(* CODESYS project sensata_utilities.library
   Company: Sensata Technologies
   Version: 1.0.2
   DocFormat: reStructuredText
   Placeholder: Sensata_Utilities
   Title: Sensata_Utilities

Project tree, tasks and I/O mapping:
  libraries: Sensata_Common, * (Sensata Technologies); Tc2_ModbusRTU, * (Beckhoff Automation GmbH); Tc2_ModbusSrv, * (Beckhoff Automation GmbH); Tc2_SerialCom, * (Beckhoff Automation GmbH); Tc2_Standard, * (Beckhoff Automation GmbH); Tc2_System, * (Beckhoff Automation GmbH); Tc2_Utilities, * (Beckhoff Automation GmbH); Tc3_JsonXml, * (Beckhoff Automation GmbH); Tc3_Module, * (Beckhoff Automation GmbH)
  Abstract/
    Obsolete/
      function block FB_DeviceAPI [ST]: M_Connect, M_Disconnect, M_GetConnectStatus, P_bConnectBusy, P_bConnected, M_CallMethod, M_GetProperty, P_bDeviceInterfaceBusy
    function block FB_CommandRouter [ST]: M_Connect, M_Disconnect, M_GetConnectStatus, P_bConnectBusy, P_bConnected, M_AwaitCommand, M_RequestRoute, M_RouteCommand, P_bCommandRoutingBusy
    function block FB_Modbus [ST]: M_Diagnostics, M_ReadCoils, M_ReadInputRegs, M_ReadInputStatus, M_ReadRegs, M_WriteMultipleCoils, M_WriteRegs, M_WriteSingleCoil, M_WriteSingleRegister, P_bModbusBusy
    function block FB_ResourceManager [ST]: M_Reset, P_bResetBusy, M_CheckIn, M_CheckOut, P_bCheckedOut, P_strCheckedOutBy
  Concrete/
    API/
      Obsolete/
        function block FB_AdsDeviceAPI [ST]: M_CallMethod, M_GetProperty, P_bDeviceInterfaceBusy
      data type E_ApiDeviceError
      function block FB_AdsCommandRouter [ST]: M_BuildMessage, M_ParseResult, M_RouteCommand, P_bCommandRoutingBusy
      function block FB_ApiDeviceTemplate [ST]: M_Abort, P_bAbortBusy, M_Connect, M_Disconnect, M_GetConnectStatus, P_bConnectBusy, P_bConnected, M_Disable, M_Enable, M_GetEnableStatus, P_bEnableBusy, P_bEnabled, M_GetPowerStatus, M_PowerOff, M_PowerOn, P_bPowerBusy, P_bPoweredOn, M_GetCurrentProgram, M_GetProgramState, M_LoadProgram, M_PauseProgram, M_StartProgram, M_StopProgram, P_bProgramControlBusy, P_enumProgramState, P_strCurrentProgram, M_Reset, P_bResetBusy, A_CommandRecovery, M_CommandTemplate, M_RouterHelper
      function block FB_ApiParamBuilder [ST]: M_AddArrayElement, M_AddEmptyArray, M_AddEmptyArrayToArray, M_AddEmptyArrayToStruct, M_AddEmptyStruct, M_AddEmptyStructToArray, M_AddEmptyStructToStruct, M_AddParameter, M_AddStructMember, M_ClearParameters, M_OutputToParameterList, M_Add, M_Pushback, M_ParseBool, M_ParseDateTime, M_ParseDouble, M_ParseInt, M_ParseInt64, M_ParseString, M_ParseUint, M_ParseUint64, M_GetArrayElement, M_GetParameter, M_GetStructMember, M_LoadFromParameterList
    IO Mapping/
      Obsolete/
        function F_LinkDigitalIOStructs [ST]
        function F_SetDigitalInput [ST]
        function F_SetDigitalOutput [ST]
        data type ST_DebugDigitalIO
      function F_LinkDigitalIO [ST]
      function F_SetDigitalIO [ST]
      data type ST_DigitalIO
    Light Control/
      function block FB_PackMLIndicators [ST]
    Modbus/
      function block FB_ModbusMasterRTU [ST]: M_Diagnostics, M_ReadCoils, M_ReadInputRegs, M_ReadInputStatus, M_ReadRegs, M_WriteMultipleCoils, M_WriteRegs, M_WriteSingleCoil, M_WriteSingleRegister, P_bModbusBusy, A_CommandRecovery
      function block FB_ModbusTCPClient [ST]: M_Diagnostics, M_ReadCoils, M_ReadInputRegs, M_ReadInputStatus, M_ReadRegs, M_WriteMultipleCoils, M_WriteRegs, M_WriteSingleCoil, M_WriteSingleRegister, P_bModbusBusy, A_CommandRecovery
    Resource Manager/
      function block FB_FifoBufferResMgr [ST]: M_Reset, P_bResetBusy, M_CheckIn, M_CheckOut, P_bCheckedOut, P_strCheckedOutBy
  DUTs/
    Obsolete/
      data type T_ApiMethodParameters
    data type E_AdsCommandRouterError
    data type ST_ApiParameter
    data type T_ApiMessage
    data type T_ApiParameterList
    data type T_ApiParamValue
  Functions/
    function F_ButtonToggle [ST]
    function F_CalcCycleTime [ST]
  Globals/
    Obsolete/
      global variables GVL_DeviceAPI
    global variables GVL_Api
  Interfaces/
    Obsolete/
      interface I_DeviceInterface: M_CallMethod, M_GetProperty, P_bDeviceInterfaceBusy
      interface I_ModularAPI: M_CallMethod, P_bApiBusy
    interface I_CommandRouting: M_AwaitCommand, M_RequestRoute, M_RouteCommand, P_bCommandRoutingBusy
    interface I_Modbus: M_ReadCoils, M_ReadInputRegs, M_ReadInputStatus, M_ReadRegs, M_WriteMultipleCoils, M_WriteRegs, M_WriteSingleCoil, M_WriteSingleRegister, P_bModbusBusy
    interface I_ResourceManagement: M_CheckIn, M_CheckOut, P_bCheckedOut, P_strCheckedOutBy
  Project Information/
    function F_GetCompany [ST]
    function F_GetTitle [ST]
    function F_GetVersion [ST]
  Version/
    global variables Global_Version
*)

// Concrete/API/E_ApiDeviceError
{attribute 'qualified_only'}
{attribute 'strict'}
TYPE E_ApiDeviceError :
(
	None := 0,
	
	CommandRouterError			:= 0100, // Error on the command router FB
	CommandFault 				:= 0101, // Command failed to execute
	
	FailedToConnect 			:= 0200, // Connect command failed
	FailedToDisconnect 			:= 0201, // Disonnect command failed
	FailedToGetConnectStatus 	:= 0202, // GetConnectStatus command failed
	
	FailedToLoadProgram			:= 0300, // LoadProgram command failed
	FailedToGetCurrentProgram	:= 0301, // GetCurrentProgram command failed
	FailedToStartProgram		:= 0302, // StartProgram command failed
	FailedToStopProgram			:= 0303, // StopProgram command failed
	FailedToPauseProgram		:= 0304, // PauseProgram command failed
	FailedToGetProgramState		:= 0305, // GetProgramState command failed
	
	FailedToEnable				:= 0400, // Enable command failed
	FailedToDisable				:= 0401, // Disable command failed
	FailedToGetEnableStatus		:= 0402, // GetEnableStatus command failed
	
	FailedToPowerOn				:= 0500, // PowerOn command failed
	FailedToPowerOff			:= 0501, // PowerOff command failed
	FailedToGetPowerStatus		:= 0502, // GetPowerStatus command failed
	
	FailedToReset				:= 0600, // Reset command failed

	FailedToAbort				:= 0700  // Abort command failed
) UDINT;
END_TYPE

// Concrete/IO Mapping/Obsolete/ST_DebugDigitalIO
{attribute 'obsolete' := 'Use ST_DigitalIO instead.'} 
TYPE ST_DebugDigitalIO :
STRUCT
	(* Label for this IO. *)
	strLabel: T_MaxString;
	(* Current value. *)
	bCurrentValue: BOOL;
	(* Set to TRUE if IO is an output. *)
	bOutput: BOOL;
	(* Set TRUE to force output to a value. *)
	bForce: BOOL;
	(* Value to force output to. *)
	bForceValue: BOOL;
END_STRUCT
END_TYPE

// Concrete/IO Mapping/ST_DigitalIO
TYPE ST_DigitalIO :
STRUCT
	(* Device this digital IO is physically connected to e.g. 'BR-100'*)
	strDevice: T_MaxString;
	(* Address of this digital IO e.g. 'Y1224' for output 1224. *)
	strAddress: T_MaxString;
	(* Label for this digital IO in English e.g. 'Tooling Down Cylinder' *)
	strLabel: T_MaxString;
	(* ID for the label for use with language switching. *)
	udintLabelId: UDINT;
	(* Current value of the digital IO. *)
	bValue: BOOL;
	(* Value to force the value to. *)
	bForceValue: BOOL;
	(* TRUE if the value is being forced. *)
	bForced: BOOL;
END_STRUCT
END_TYPE

// DUTs/Obsolete/T_ApiMethodParameters
{attribute 'obsolete' := 'Only used on obsolete FB_DeviceAPI'} 
TYPE T_ApiMethodParameters : 
	ARRAY [1..GVL_DeviceAPI.uintMAX_CALL_METHOD_PARAMETERS]
		OF ARRAY [1..2] OF Tc2_System.T_MaxString;
END_TYPE

// DUTs/E_AdsCommandRouterError
{attribute 'qualified_only'}
{attribute 'strict'}
TYPE E_AdsCommandRouterError :
(
	None := 0,
	IncorrectResponseFormat := 100,
	NoResponseReceived := 101,
	AdsError := 200,
	PointerError := 300
) UDINT;
END_TYPE

// DUTs/ST_ApiParameter
TYPE ST_ApiParameter :
STRUCT
	strKey : T_MaxString;
	strValue : T_ApiParamValue;
END_STRUCT
END_TYPE

// DUTs/T_ApiMessage
TYPE T_ApiMessage : STRING(GVL_Api.dintMSG_STRING_SIZE); END_TYPE

// DUTs/T_ApiParameterList
TYPE T_ApiParameterList : ARRAY[GVL_Api.dintPARAM_LOWER_BOUND..GVL_Api.dintPARAM_UPPER_BOUND] OF ST_ApiParameter; END_TYPE

// DUTs/T_ApiParamValue
TYPE T_ApiParamValue : STRING(GVL_Api.dintPARAM_STRING_SIZE); END_TYPE

// Globals/Obsolete/GVL_DeviceAPI
{attribute 'qualified_only'}
VAR_GLOBAL CONSTANT
	uintMAX_CALL_METHOD_PARAMETERS : UINT := 16;
END_VAR

// Globals/GVL_Api
{attribute 'qualified_only'}
VAR_GLOBAL CONSTANT
	dintPARAM_LOWER_BOUND : DINT := 0;
	dintPARAM_UPPER_BOUND : DINT := 31;
	dintPARAM_STRING_SIZE : DINT := 1023;
	dintMSG_STRING_SIZE : DINT := 4095;
END_VAR

// Version/Global_Version
{attribute 'TcGenerated'}
{attribute 'no-analysis'}
{attribute 'linkalways'}
// This function has been automatically generated from the project information.
VAR_GLOBAL CONSTANT
	{attribute 'const_non_replaced'}
	stLibVersion_Sensata_Utilities : ST_LibVersion := (iMajor := 1, iMinor := 0, iBuild := 2, iRevision := 0, nFlags := 0, sVersion := '1.0.2');
END_VAR

// Abstract/Obsolete/FB_DeviceAPI
(*
===============================================================================
Abstract Device API
===============================================================================
:Contact: Kevin Sanita <ksanita@sensata.com>
:Last Edited: March 2022

:Description: Represents a device API that allows for methods and
	properties to be called and accessed

:Notes:
* ``M_CallMethod`` to send a call method command to a device API
* ``M_GetProperty`` to send a get property command to a device API

:Change Log:
- **March 25, 2022** Initial version
*)
{attribute 'obsolete' := 'Use FB_CommandRouter instead!'} 
FUNCTION_BLOCK ABSTRACT FB_DeviceAPI EXTENDS FB_Module IMPLEMENTS I_DeviceInterface, I_Connectable
VAR_INPUT
END_VAR
VAR_OUTPUT
END_VAR
VAR
	bConnected: BOOL;
END_VAR

(* Connect to the device. *)
METHOD M_Connect : BOOL
bConnected := TRUE;
M_Connect := TRUE;
THIS^.M_LogWarning('M_Connect not implemented!');
END_METHOD

(* Disconnect from the camera. *)
METHOD M_Disconnect : BOOL
bConnected := FALSE;
M_Disconnect := TRUE;
THIS^.M_LogWarning('M_Disconnect not implemented!');
END_METHOD

(* Get the device connection status. *)
METHOD M_GetConnectStatus : BOOL
VAR_OUTPUT
	(* TRUE if the device is connected, FALSE otherwise. *)
	bConnected	: BOOL;
END_VAR
bConnected := THIS^.bConnected;
M_GetConnectStatus := TRUE;
END_METHOD

(* TRUE while the device is connecting or disconnecting. *)
PROPERTY P_bConnectBusy : BOOL
GET
P_bConnectBusy := FALSE;
END_GET
END_PROPERTY

(* TRUE if the camera is connected. *)
PROPERTY P_bConnected : BOOL
GET
P_bConnected := bConnected;
END_GET
END_PROPERTY

(* Calls a device method from a device API. *)
METHOD M_CallMethod : BOOL
VAR_INPUT
	(* UniqueID of the target module. *)
	strTargetId		: Tc2_System.T_MaxString;
	(* Name of the method to call. *)
	strMethodName	: Tc2_System.T_MaxString;
	(* 2D array of parameter name and parameter value. *)
	arrParameters	: T_ApiMethodParameters;
END_VAR
VAR_OUTPUT
	(* Return data of the method. *)
	strReturn	: Tc2_System.T_MaxString;
END_VAR
M_CallMethod := FALSE;
END_METHOD

(* Gets the value of a device property through an API. *)
METHOD M_GetProperty : BOOL
VAR_INPUT
	(* Name of the property to get. *)
	strPropertyName	: Tc2_System.T_MaxString;
END_VAR
VAR_OUTPUT
	(* Value of the property. *)
	strReturn	: Tc2_System.T_MaxString;
END_VAR
M_GetProperty := FALSE;
END_METHOD

(* True while a device interface command is running. *)
PROPERTY P_bDeviceInterfaceBusy : BOOL
GET
P_bDeviceInterfaceBusy := FALSE;
END_GET
END_PROPERTY

END_FUNCTION_BLOCK

// Abstract/FB_CommandRouter
FUNCTION_BLOCK FB_CommandRouter EXTENDS FB_Module
	IMPLEMENTS I_CommandRouting, I_Connectable
VAR_INPUT
END_VAR
VAR_OUTPUT
END_VAR
VAR
	cr_bConnected: BOOL;
END_VAR

(* This method should establish any external connections required to use the
	functions of the device, and return TRUE and set P_bConnected to TRUE once
	connected. *)
METHOD M_Connect : BOOL
THIS^.M_LogWarning('M_Connect not implemented!');
cr_bConnected := TRUE;
M_Connect := TRUE;
END_METHOD

(* This method should break any connections established by M_Connect. It should
	immediately set P_bConnected to false unless all connections are known to
	be still active, and return TRUE once those connections are all fully
	disconnected. *)
METHOD M_Disconnect : BOOL
THIS^.M_LogWarning('M_Disconnect not implemented!');
cr_bConnected := FALSE;
M_Disconnect := TRUE;
END_METHOD

(* This method should explicitly check the connection status of the device.
	Once the connection status is known, this method should return TRUE.
	If this method fails, P_bConnected should be set to FALSE since the device
	is not absolutely known to still be connected. *)
METHOD M_GetConnectStatus : BOOL
VAR_OUTPUT
	(* This should return TRUE if all connections required to make the device
		function properly are known to be connected, and FALSE otherwise. *)
	bConnected	: BOOL;
END_VAR
THIS^.M_LogWarning('M_GetConnectStatus not implemented!');
M_GetConnectStatus := TRUE;
bConnected := cr_bConnected;
END_METHOD

(* This property should be TRUE while any method in this interface is actively
	executing, or FALSE otherwise. *)
PROPERTY P_bConnectBusy : BOOL
GET
P_bConnectBusy := FALSE;
END_GET
END_PROPERTY

(* This should be set to TRUE if M_Connect is successful or M_GetConnectStatus
	determines the device to be connected, and set to FALSE if M_Disconnect is
	called at all, M_GetConnectStatus fails, or M_GetConnectStatus determines
	the device to be not connected. *)
PROPERTY P_bConnected : BOOL
GET
P_bConnected := cr_bConnected;
END_GET
END_PROPERTY

(* Waits for the command with the given route ID to complete. *)
METHOD M_AwaitCommand : BOOL
VAR_INPUT
	(* ID assigned to the route. *)
	_in_udintRouteId	: UDINT;
	(* Timeout time for the command. *)
	_in_timeTimeout	: TIME;
END_VAR
VAR_IN_OUT
	(* Array of data key:value pairs. This will be filled with output
		data on command success. This is required due to memory limitations
		within Beckhoff. *)
	_inout_arrOutputs	: T_ApiParameterList;
END_VAR
VAR_OUTPUT
	(* True if the command executed without error. Does not necessarily
	mean the command performed the task it was expected to perform, just
	means that the method returned a value. *)
	_out_bCommandExecuted	: BOOL;
	(* The return value of the method. *)
	_out_strReturnValue	: T_ApiParamValue;
END_VAR
THIS^.M_LogWarning('M_AwaitCommand not implemented!');
M_AwaitCommand := TRUE;
END_METHOD

(* Sends a route request and returns a route ID if successfully routed. 
Use M_AwaitCommand with the route ID as input in order to wait for and get
the results of the routed command. *)
METHOD M_RequestRoute : BOOL
VAR_INPUT
	(* Unique ID of the module to call the command on. *)
	_in_strModuleId	: Tc2_System.T_MaxString;
	(* Name of the method to call. *)
	_in_strMethodName	: Tc2_System.T_MaxString;
	(* Timeout time for the route. *)
	_in_timeTimeout	: TIME;
END_VAR
VAR_IN_OUT
	(* Array of data key:value pairs. This should be set to the parameters
		of the command. *)
	_inout_arrParameters	: T_ApiParameterList;
END_VAR
VAR_OUTPUT
	(* ID assigned to the route. *)
	_out_udintRouteId	: UDINT;
END_VAR
THIS^.M_LogWarning('M_RequestRoute not implemented!');
M_RequestRoute := TRUE;
END_METHOD

(* Routes the given command and waits for the command to finish before
returning the output data of the command. *)
METHOD M_RouteCommand : BOOL
VAR_INPUT
	(* Unique ID of the module to call the command on. *)
	_in_strModuleId	: Tc2_System.T_MaxString;
	(* Name of the method to call. *)
	_in_strMethodName	: Tc2_System.T_MaxString;
	(* Timeout time for the command. *)
	_in_timeTimeout	: TIME;
END_VAR
VAR_IN_OUT
	(* Array of input parameter key:value pairs. *)
	_inout_arrParameters	: T_ApiParameterList;
	(* Array of output key:value pairs. Will be cleared and then populated with output data. *)
	_inout_arrOutputs	: T_ApiParameterList;
END_VAR
VAR_OUTPUT
	(* True if the command executed without error. Does not necessarily
	mean the command performed the task it was expected to perform, just
	means that the method returned a value. *)
	_out_bCommandExecuted	: BOOL;
	(* The return value of the method as a string. *)
	_out_strReturnValue	: T_ApiParamValue;
END_VAR
THIS^.M_LogWarning('M_RouteCommand not implemented!');
M_RouteCommand := TRUE;
END_METHOD

(* TRUE while any method in this interface is running. *)
PROPERTY P_bCommandRoutingBusy : BOOL
GET
P_bCommandRoutingBusy := TRUE;
END_GET
END_PROPERTY

END_FUNCTION_BLOCK

// Interfaces/I_CommandRouting
INTERFACE I_CommandRouting

(* Waits for the command with the given route ID to complete. *)
METHOD M_AwaitCommand : BOOL
VAR_INPUT
	(* ID assigned to the route. *)
	_in_udintRouteId : UDINT;
	
	(* Timeout time for the command. *)
	_in_timeTimeout : TIME;
END_VAR
VAR_IN_OUT
	(* Array of data key:value pairs. This will be filled with output
		data on command success. This is required due to memory limitations
		within Beckhoff. *)
	_inout_arrOutputs : T_ApiParameterList;
END_VAR
VAR_OUTPUT
	(* True if the command executed without error. Does not necessarily
	mean the command performed the task it was expected to perform, just
	means that the method returned a value. *)
	_out_bCommandExecuted : BOOL;
	
	(* The return value of the method. *)
	_out_strReturnValue : T_ApiParamValue;
END_VAR
END_METHOD

(* Sends a route request and returns a route ID if successfully routed. 
Use M_AwaitCommand with the route ID as input in order to wait for and get
the results of the routed command. *)
METHOD M_RequestRoute : BOOL
VAR_INPUT
	(* Unique ID of the module to call the command on. *)
	_in_strModuleId : T_MaxString;
	
	(* Name of the method to call. *)
	_in_strMethodName : T_MaxString;
	
	(* Timeout time for the route. *)
	_in_timeTimeout : TIME;
END_VAR
VAR_IN_OUT
	(* Array of data key:value pairs. This should be set to the parameters
		of the command. *)
	_inout_arrParameters : T_ApiParameterList;
END_VAR
VAR_OUTPUT
	(* ID assigned to the route. *)
	_out_udintRouteId : UDINT;
END_VAR
END_METHOD

(* Routes the given command and waits for the command to finish before
returning the output data of the command. *)
METHOD M_RouteCommand : BOOL
VAR_INPUT
	(* Unique ID of the module to call the command on. *)
	_in_strModuleId	: Tc2_System.T_MaxString;
	
	(* Name of the method to call. *)
	_in_strMethodName	: Tc2_System.T_MaxString;
	
	(* Timeout time for the command. *)
	_in_timeTimeout	: TIME;
END_VAR
VAR_IN_OUT
	(* Array of input parameter key:value pairs. *)
	_inout_arrParameters	: T_ApiParameterList;
	
	(* Array of output key:value pairs. Will be cleared and then populated with output data. *)
	_inout_arrOutputs	: T_ApiParameterList;
END_VAR
VAR_OUTPUT
	(* True if the command executed without error. Does not necessarily
	mean the command performed the task it was expected to perform, just
	means that the method returned a value. *)
	_out_bCommandExecuted	: BOOL;
	
	(* The return value of the method as a string. *)
	_out_strReturnValue	: T_ApiParamValue;
END_VAR
END_METHOD

(* TRUE while any method in this interface is running. *)
PROPERTY P_bCommandRoutingBusy : BOOL
GET
END_GET
END_PROPERTY

END_INTERFACE

// Interfaces/Obsolete/I_DeviceInterface
INTERFACE I_DeviceInterface

(* Calls a device method from a device API. *)
METHOD M_CallMethod : BOOL
VAR_INPUT
	(* UniqueID of the target module. *)
	strTargetId		: Tc2_System.T_MaxString;
		
	(* Name of the method to call. *)
	strMethodName : T_MaxString;
	
	(* 2D array of parameter name and parameter value. *)
	arrParameters : T_ApiMethodParameters;
END_VAR
VAR_OUTPUT
	(* Return data of the method. *)
	strReturn : T_MaxString;
END_VAR
END_METHOD

(* Gets the value of a device property through an API. *)
METHOD M_GetProperty : BOOL
VAR_INPUT
	(* Name of the property to get. *)
	strPropertyName : T_MaxString;
END_VAR
VAR_OUTPUT
	(* Value of the property. *)
	strReturn : T_MaxString;
END_VAR
END_METHOD

(* True while a device interface command is running. *)
PROPERTY P_bDeviceInterfaceBusy : BOOL
GET
END_GET
END_PROPERTY

END_INTERFACE

// Abstract/FB_Modbus
FUNCTION_BLOCK ABSTRACT FB_Modbus EXTENDS FB_Module
	IMPLEMENTS I_Modbus
VAR_INPUT
END_VAR
VAR_OUTPUT
END_VAR
VAR
END_VAR

(* Modbus Function Code 8 = Diagnostic *)
(* The diagnosis function provides a series of tests for checking the communication 
system between the master and the slave and for examining a variety of internal 
error states within the slave *)
METHOD M_Diagnostics : BOOL
VAR_INPUT
	(* Timeout value for waiting for a response from the addressed slave *)
	_in_timeTimeout : TIME;	
END_VAR
VAR_OUTPUT
	(* Contains the number of bytes currently read *)
	_out_udintcbRead : UDINT;
END_VAR
M_Diagnostics := TRUE;
THIS^.M_LogWarning('M_Diagnostics not implemented!');
END_METHOD

(* Modbus Function Code 1 = Read Coils *)
(* This function is used for reading 1 to 2048 digital outputs (coils.
One digital output corresponds to one bit of the read data bytes. *)
METHOD M_ReadCoils : BOOL
VAR_INPUT
	(* Number of data words to be read or written for word-oriented Modbus functions. For bit-oriented Modbus functions, Quantity specifies the number of bits (inputs or coils) *)
	_in_wordQuantity : WORD;
	(* Modbus Data Address from which the data are read from the end device(slave) *)
	_in_wordMBAddr : WORD;
	(* Size of the data variable used for send or read actions in bytes *)
	_in_udintcbLength : UDINT;
	(* pDestAddr for Modbus TCP FB_MBReadCoils*)
	_in_bytepMemoryAddr	: POINTER TO BYTE;
	(* Timeout value for waiting for a response from the addressed slave *)
	_in_timeTimeout	: TIME;
END_VAR
VAR_OUTPUT
	(* Contains the number of bytes currently read *)
	_out_udintcbRead : UDINT;
END_VAR
M_ReadCoils := TRUE;
THIS^.M_LogWarning('M_ReadCoils not implemented!');
END_METHOD

(* Modbus Function Code 4 = Read Input Registers *)
(* This function is used for reading 1 to 128 output registers (16 bit.
The first byte contains the lower eight bits and the second byte the upper eight bits. *)
METHOD M_ReadInputRegs : BOOL
VAR_INPUT
	(* Number of data words to be read or written for word-oriented Modbus functions. For bit-oriented Modbus functions, Quantity specifies the number of bits (inputs or coils) *)
	_in_wordQuantity : WORD;
	(* Modbus Data Address from which the data are read from the end device(slave) *)
	_in_wordMBAddr : WORD;
	(* Size of the data variable used for send or read actions in bytes *)
	_in_udintcbLength : UDINT;
	(* pDestAddr for Modbus TCP FB_MBReadInputRegs*)
	_in_bytepMemoryAddr : POINTER TO BYTE;
	(* Timeout value for waiting for a response from the addressed slave *)
	_in_timeTimeout : TIME;
END_VAR
VAR_OUTPUT
	(* Contains the number of bytes currently read *)
	_out_udintcbRead : UDINT;
END_VAR
M_ReadInputRegs := TRUE;
THIS^.M_LogWarning('M_ReadInputRegs not implemented!');
END_METHOD

(* Modbus Function Code 2 = Read Discrete Inputs *)
(* This function is used for reading 1 to 2048 digital inputs. One digital input 
corresponds to one bit of the read data bytes *)
METHOD M_ReadInputStatus : BOOL (* FB_MBReadInputs for Modbus TCP*)
VAR_INPUT
	(* Number of data words to be read or written for word-oriented Modbus functions. For bit-oriented Modbus functions, Quantity specifies the number of bits (inputs or coils) *)
	_in_wordQuantity : WORD;
	(* Modbus Data Address from which the data are read from the end device(slave) *)
	_in_wordMBAddr	: WORD;
	(* Size of the data variable used for send or read actions in bytes *)
	_in_udintcbLength : UDINT;
	(* pDestAddr for Modbus TCP FB_MBReadInputs*)
	_in_bytepMemoryAddr	: POINTER TO BYTE;
	(* Timeout value for waiting for a response from the addressed slave *)
	_in_timeTimeout	: TIME;
END_VAR
VAR_OUTPUT
	(* Contains the number of bytes currently read *)
	_out_udintcbRead : UDINT;
END_VAR
M_ReadInputStatus := TRUE;
THIS^.M_LogWarning('M_ReadInputStatus not implemented!');
END_METHOD

(* Modbus Function Code 3 = Read Registers *)
(* This function is used for reading 1 to 128 output registers (16 bit). 
The first byte contains the lower eight bits and the second byte the upper eight bits. *)
METHOD M_ReadRegs : BOOL
VAR_INPUT
	(* Number of data words to be read or written for word-oriented Modbus functions. For bit-oriented Modbus functions, Quantity specifies the number of bits (inputs or coils) *)
	_in_wordQuantity : WORD;
	(* Modbus Data Address from which the data are read from the end device(slave) *)
	_in_wordMBAddr : WORD;
	(* Size of the data variable used for send or read actions in bytes *)
	_in_udintcbLength : UDINT;
	(* pDestAddr for Modbus TCP FB_MBReadRegs*)
	_in_bytepMemoryAddr	: POINTER TO BYTE;
	(* Timeout value for waiting for a response from the addressed slave *)
	_in_timeTimeout	: TIME;
END_VAR
VAR_OUTPUT
	(* Contains the number of bytes currently read *)
	_out_udintcbRead : UDINT;
END_VAR
M_ReadRegs := TRUE;
THIS^.M_LogWarning('M_ReadRegs not implemented!');
END_METHOD

(* Modbus Function Code 15 = Write Multiple Coils *)
(* This function is used for writing 1 to 2048 digital outputs (coils). 
One digital output corresponds to one bit of the write data bytes *)
METHOD M_WriteMultipleCoils : BOOL (* FB_MBWriteCoils for Modbus TCP*)
VAR_INPUT
	(* Number of data words to be read or written for word-oriented Modbus functions. For bit-oriented Modbus functions, Quantity specifies the number of bits (inputs or coils) *)
	_in_wordQuantity : WORD;
	(* Modbus Data Address from which the data are read from the end device(slave) *)
	_in_wordMBAddr : WORD;
	(* Size of the data variable used for send or read actions in bytes *)
	_in_udintcbLength : UDINT;
	(* pDestAddr for Modbus TCP FB_MBReadCoils*)
	_in_bytepMemoryAddr	: POINTER TO BYTE;
	(* Timeout value for waiting for a response from the addressed slave *)
	_in_timeTimeout	: TIME;
END_VAR
M_WriteMultipleCoils := TRUE;
THIS^.M_LogWarning('M_WriteMultipleCoils not implemented!');
END_METHOD

(* Modbus Function Code 16 = Write Registers *)
(* This function is used for writing 1 to 128 output registers (16 bit). *)
METHOD M_WriteRegs : BOOL
VAR_INPUT
	(* Number of data words to be read or written for word-oriented Modbus functions. For bit-oriented Modbus functions, Quantity specifies the number of bits (inputs or coils) *)
	_in_wordQuantity : WORD;
	(* Modbus Data Address from which the data are read from the end device(slave) *)
	_in_wordMBAddr	: WORD;
	(* Size of the data variable used for send or read actions in bytes *)
	_in_udintcbLength : UDINT;
	(* pDestAddr for Modbus TCP FB_MBWriteRegs*)
	_in_bytepMemoryAddr	: POINTER TO BYTE;
	(* Timeout value for waiting for a response from the addressed slave *)
	_in_timeTimeout	: TIME;
END_VAR
M_WriteRegs := TRUE;
THIS^.M_LogWarning('M_WriteRegs not implemented!');
END_METHOD

(* Modbus Function Code 5 = Write Single Coil *)
(* This function is used for writing a single digital output (coil). Bit access is used. *)
METHOD M_WriteSingleCoil : BOOL
VAR_INPUT
	(* Modbus Data Address from which the data are read from the end device(slave) *)
	_in_wordMBAddr : WORD;
	(* Value to be written into the digital output. Method parses boolean "TRUE" to 16#FF00 to switch the output on, and boolean "FALSE" to 16#0000 to switch it off. *)
	_in_bValue : BOOL;
	(* Timeout value for waiting for a response from the addressed slave *)
	_in_timeTimeout	: TIME;
END_VAR
M_WriteSingleCoil := TRUE;
THIS^.M_LogWarning('M_WriteSingleCoil not implemented!');
END_METHOD

(* Modbus Function Code 6 = Write Single Register *)
(* This function is used for writing an individual output register. 16 bit access is used. *)
METHOD M_WriteSingleRegister : BOOL
VAR_INPUT
	(* Modbus Data Address from which the data are read from the end device(slave) *)
	_in_wordMBAddr : WORD;
	(* Value to be written into the register (word value) *)
	_in_nValue : WORD;
	(* Timeout value for waiting for a response from the addressed slave *)
	_in_timeTimeout	: TIME;
END_VAR
M_WriteSingleRegister := TRUE;
THIS^.M_LogWarning('M_WriteSingleRegister not implemented!');
END_METHOD

(* This property should be TRUE while any method in this interface is actively
	executing, or FALSE otherwise. *)
PROPERTY P_bModbusBusy : BOOL
GET
P_bModbusBusy := FALSE;
END_GET
END_PROPERTY

END_FUNCTION_BLOCK

// Interfaces/I_Modbus
(*
===============================================================================
Modbus
===============================================================================

:Description: Interface that implements the ability for Modbus communications
   as RTU Master or TCP Client mode.

*)

INTERFACE I_Modbus

(* Modbus Function Code 1 = Read Coils *)
(* This function is used for reading 1 to 2048 digital outputs (coils.
One digital output corresponds to one bit of the read data bytes. *)
METHOD M_ReadCoils : BOOL
VAR_INPUT
	(* Number of data words to be read or written for word-oriented Modbus functions. For bit-oriented Modbus functions, Quantity specifies the number of bits (inputs or coils) *)
	_in_wordQuantity : WORD;
	(* Modbus Data Address from which the data are read from the end device(slave) *)
	_in_wordMBAddr : WORD;
	(* Size of the data variable used for send or read actions in bytes *)
	_in_udintcbLength : UDINT;
	(* Memory address in the PLC, calculated with ADR (Modbus data) *)
	_in_bytepMemoryAddr : POINTER TO BYTE;  // pDestAddr for Modbus TCP FB_MBReadCoils
	(* Timeout value for waiting for a response from the addressed slave *)
	_in_timeTimeout : TIME;	
END_VAR
VAR_OUTPUT
	(* Contains the number of bytes currently read *)
	_out_udintcbRead : UDINT;
END_VAR
END_METHOD

(* Modbus Function Code 4 = Read Input Registers *)
(* This function is used for reading 1 to 128 output registers (16 bit.
The first byte contains the lower eight bits and the second byte the upper eight bits. *)
METHOD M_ReadInputRegs : BOOL
VAR_INPUT
	(* Number of data words to be read or written for word-oriented Modbus functions. For bit-oriented Modbus functions, Quantity specifies the number of bits (inputs or coils) *)
	_in_wordQuantity : WORD;
	(* Modbus Data Address from which the data are read from the end device(slave) *)
	_in_wordMBAddr : WORD;
	(* Size of the data variable used for send or read actions in bytes *)
	_in_udintcbLength : UDINT;
	(* Memory address in the PLC, calculated with ADR (Modbus data) *)
	_in_bytepMemoryAddr : POINTER TO BYTE;  // pDestAddr for Modbus TCP FB_MBReadInputRegs
	(* Timeout value for waiting for a response from the addressed slave *)
	_in_timeTimeout : TIME;	
END_VAR
VAR_OUTPUT
	(* Contains the number of bytes currently read *)
	_out_udintcbRead : UDINT;
END_VAR
END_METHOD

(* Modbus Function Code 2 = Read Discrete Inputs *)
(* This function is used for reading 1 to 2048 digital inputs. One digital input 
corresponds to one bit of the read data bytes *)
METHOD M_ReadInputStatus : BOOL (* FB_MBReadInputs for Modbus TCP*)
VAR_INPUT
	(* Number of data words to be read or written for word-oriented Modbus functions. For bit-oriented Modbus functions, Quantity specifies the number of bits (inputs or coils) *)
	_in_wordQuantity : WORD;
	(* Modbus Data Address from which the data are read from the end device(slave) *)
	_in_wordMBAddr : WORD;
	(* Size of the data variable used for send or read actions in bytes *)
	_in_udintcbLength : UDINT;
	(* Memory address in the PLC, calculated with ADR (Modbus data) *)
	_in_bytepMemoryAddr : POINTER TO BYTE;  // pDestAddr for Modbus TCP FB_MBReadInputs
	(* Timeout value for waiting for a response from the addressed slave *)
	_in_timeTimeout : TIME;	
END_VAR
VAR_OUTPUT
	(* Contains the number of bytes currently read *)
	_out_udintcbRead : UDINT;
END_VAR
END_METHOD

(* Modbus Function Code 3 = Read Registers *)
(* This function is used for reading 1 to 128 output registers (16 bit). 
The first byte contains the lower eight bits and the second byte the upper eight bits. *)
METHOD M_ReadRegs : BOOL
VAR_INPUT
	(* Number of data words to be read or written for word-oriented Modbus functions. For bit-oriented Modbus functions, Quantity specifies the number of bits (inputs or coils) *)
	_in_wordQuantity : WORD;
	(* Modbus Data Address from which the data are read from the end device(slave) *)
	_in_wordMBAddr : WORD;
	(* Size of the data variable used for send or read actions in bytes *)
	_in_udintcbLength : UDINT;
	(* Memory address in the PLC, calculated with ADR (Modbus data) *)
	_in_bytepMemoryAddr : POINTER TO BYTE;  // pDestAddr for Modbus TCP FB_MBReadRegs
	(* Timeout value for waiting for a response from the addressed slave *)
	_in_timeTimeout : TIME;	
END_VAR
VAR_OUTPUT
	(* Contains the number of bytes currently read *)
	_out_udintcbRead : UDINT;
END_VAR
END_METHOD

(* Modbus Function Code 15 = Write Multiple Coils *)
(* This function is used for writing 1 to 2048 digital outputs (coils). 
One digital output corresponds to one bit of the write data bytes *)
METHOD M_WriteMultipleCoils : BOOL (* FB_MBWriteCoils for Modbus TCP*)
VAR_INPUT
	(* Number of data words to be read or written for word-oriented Modbus functions. For bit-oriented Modbus functions, Quantity specifies the number of bits (inputs or coils) *)
	_in_wordQuantity : WORD;
	(* Modbus Data Address from which the data are read from the end device(slave) *)
	_in_wordMBAddr : WORD;
	(* Size of the data variable used for send or read actions in bytes *)
	_in_udintcbLength : UDINT;
	(* Memory address in the PLC, calculated with ADR (Modbus data) *)
	_in_bytepMemoryAddr : POINTER TO BYTE;  // pDestAddr for Modbus TCP FB_MBReadCoils
	(* Timeout value for waiting for a response from the addressed slave *)
	_in_timeTimeout : TIME;	
END_VAR
END_METHOD

(* Modbus Function Code 16 = Write Registers *)
(* This function is used for writing 1 to 128 output registers (16 bit). *)
METHOD M_WriteRegs : BOOL
VAR_INPUT
	(* Number of data words to be read or written for word-oriented Modbus functions. For bit-oriented Modbus functions, Quantity specifies the number of bits (inputs or coils) *)
	_in_wordQuantity : WORD;
	(* Modbus Data Address from which the data are read from the end device(slave) *)
	_in_wordMBAddr : WORD;
	(* Size of the data variable used for send or read actions in bytes *)
	_in_udintcbLength : UDINT;
	(* Memory address in the PLC, calculated with ADR (Modbus data) *)
	_in_bytepMemoryAddr : POINTER TO BYTE;  // pDestAddr for Modbus TCP FB_MBWriteRegs
	(* Timeout value for waiting for a response from the addressed slave *)
	_in_timeTimeout : TIME;	
END_VAR
END_METHOD

(* Modbus Function Code 5 = Write Single Coil *)
(* This function is used for writing a single digital output (coil). Bit access is used. *)
METHOD M_WriteSingleCoil : BOOL
VAR_INPUT
	(* Modbus Data Address from which the data are read from the end device(slave) *)
	_in_wordMBAddr : WORD;
	(* Value to be written into the digital output. Method parses boolean "TRUE" to 16#FF00 to switch the output on, and boolean "FALSE" to 16#0000 to switch it off. *)
	_in_bValue : BOOL;
	(* Timeout value for waiting for a response from the addressed slave *)
	_in_timeTimeout : TIME;
END_VAR
END_METHOD

(* Modbus Function Code 6 = Write Single Register *)
(* This function is used for writing an individual output register. 16 bit access is used. *)
METHOD M_WriteSingleRegister : BOOL
VAR_INPUT
	(* Modbus Data Address from which the data are read from the end device(slave) *)
	_in_wordMBAddr : WORD;
	(* Value to be written into the register (word value) *)
	_in_nValue : WORD;
	(* Timeout value for waiting for a response from the addressed slave *)
	_in_timeTimeout : TIME;	
END_VAR
END_METHOD

(* This property should be TRUE while any method in this interface is actively
	executing, or FALSE otherwise. *)
PROPERTY P_bModbusBusy : BOOL
GET
END_GET
END_PROPERTY

END_INTERFACE

// Abstract/FB_ResourceManager
(* FB to manage a shared resource. *)
FUNCTION_BLOCK ABSTRACT FB_ResourceManager EXTENDS FB_Module IMPLEMENTS I_ResourceManagement, I_Resettable
VAR_INPUT
END_VAR
VAR_OUTPUT
END_VAR
VAR
	rm_strCheckedOutBy: T_MaxString;
END_VAR

(* This should clear any errors on the device and bring it to a state where
	it is ready to be energized or otherwise activated. *)
METHOD M_Reset : BOOL
THIS^.M_LogWarning('M_Reset not implemented!');
M_Reset := TRUE;
END_METHOD

(* This property should be TRUE while any method in this interface is actively
	executing, or FALSE otherwise. *)
PROPERTY P_bResetBusy : BOOL
GET
P_bResetBusy := FALSE;
END_GET
END_PROPERTY

(* Checks in the resource for the given module. *)
METHOD M_CheckIn : BOOL
VAR_INPUT
	(* ID of the module checking the resource out. *)
	_in_strId	: Tc2_System.T_MaxString;
END_VAR
rm_strCheckedOutBy := '';
THIS^.M_LogWarning('M_CheckIn not implemented!');
M_CheckIn := TRUE;
END_METHOD

(* Checks out the resource for the given module ID. *)
METHOD M_CheckOut : BOOL
VAR_INPUT
	(* ID of the module checking the resource out. *)
	_in_strId	: Tc2_System.T_MaxString;
END_VAR
rm_strCheckedOutBy := _in_strId;
THIS^.M_LogWarning('M_CheckOut not implemented!');
M_CheckOut := TRUE;
END_METHOD

(* TRUE if the resource is checked out. *)
PROPERTY P_bCheckedOut : BOOL
GET
P_bCheckedOut := LEN(rm_strCheckedOutBy) > 0;
END_GET
END_PROPERTY

(* ID of the module checking out the resource. *)
PROPERTY P_strCheckedOutBy : Tc2_System.T_MaxString
GET
P_strCheckedOutBy := rm_strCheckedOutBy;
END_GET
END_PROPERTY

END_FUNCTION_BLOCK

// Interfaces/I_ResourceManagement
INTERFACE I_ResourceManagement

(* Checks in the resource for the given module. *)
METHOD M_CheckIn : BOOL
VAR_INPUT
	(* ID of the module checking the resource out. *)
	_in_strId: T_MaxString;
END_VAR
END_METHOD

(* Checks out the resource for the given module ID. *)
METHOD M_CheckOut : BOOL
VAR_INPUT
	(* ID of the module checking the resource out. *)
	_in_strId: T_MaxString;
END_VAR
END_METHOD

(* TRUE if the resource is checked out. *)
PROPERTY P_bCheckedOut : BOOL
GET
END_GET
END_PROPERTY

(* ID of the module checking out the resource. *)
PROPERTY P_strCheckedOutBy : T_MaxString
GET
END_GET
END_PROPERTY

END_INTERFACE

// Concrete/API/Obsolete/FB_AdsDeviceAPI
(*
===============================================================================
ADS Device API
===============================================================================
:Contact: Kevin Sanita <ksanita@sensata.com>
:Last Edited: March 2022

:Description: Represents a device API that allows for methods and
	properties to be called and accessed through ADS

:Notes:
* ``M_CallMethod`` to send a call method command to a device API through ADS
* ``M_GetProperty`` to send a get property command to a device API through ADS

:Change Log:
- **March 25, 2022** Initial version
*)
{attribute 'obsolete' := 'Use FB_AdsCommandRouter instead!'} 
FUNCTION_BLOCK FB_AdsDeviceAPI EXTENDS FB_DeviceAPI IMPLEMENTS I_DeviceInterface
VAR_INPUT
	(* ADS address of the device ADS server. *)
	strAdsAddress: T_AmsNetId;
	
	(* ADS port of the device ADS server. *)
	udintAdsPort: T_AmsPort;
	
	(* Optional timeout for the ADS commands. Default 60 seconds. *)
	timeAdsTimeout: TIME := T#60S;
END_VAR
VAR_OUTPUT
END_VAR
VAR CONSTANT
	udintGET_PROPERTY_GROUP : UDINT := 16#1000;
	udintGET_PROPERTY_OFFSET : UDINT := 0;
	udintCALL_METHOD_GROUP : UDINT := 16#2000;
	udintCALL_METHOD_OFFSET : UDINT := 0;
END_VAR
VAR
	fbAds: ADSRDWRTEX;
	udintGroup: UDINT;
	udintOffset: UDINT;
	strMessage: T_MaxString;
	bSend: BOOL;
	udintAdsReadByteCount: UDINT;
	strResponse: T_MaxString;
	bAdsBusy: BOOL;
	udintAdsErrorId: UDINT;
	bBusy: BOOL;
	bAdsError: BOOL;
	fbJson: FB_JsonDomParser;
	intCallMethodStep: INT;
	intGetPropertyStep: INT;
END_VAR

fbAds(
	NETID:= strAdsAddress, 
	PORT:= udintAdsPort, 
	IDXGRP:= udintGroup, 
	IDXOFFS:= udintOffset, 
	WRITELEN:= INT_TO_UDINT(LEN(strMessage)), 
	READLEN:= SIZEOF(T_MaxString), 
	SRCADDR:= ADR(strMessage), 
	DESTADDR:= ADR(strResponse), 
	WRTRD:= bSend, 
	TMOUT:= timeAdsTimeout, 
	BUSY=> bAdsBusy, 
	ERR=> bAdsError, 
	ERRID=> udintAdsErrorId, 
	COUNT_R=> udintAdsReadByteCount);
	
bSend := FALSE;

(* Calls a device method from a device API. *)
METHOD M_CallMethod : BOOL
VAR_INPUT
	(* UniqueID of the target module. *)
	strTargetId		: Tc2_System.T_MaxString;
	(* Name of the method to call. *)
	strMethodName	: Tc2_System.T_MaxString;
	(* 2D array of parameter name and parameter value. *)
	arrParameters	: T_ApiMethodParameters;
END_VAR
VAR_OUTPUT
	(* Return data of the method. *)
	strReturn	: Tc2_System.T_MaxString;
END_VAR

VAR
	strCommand : T_MaxString;
	jsonParams: Tc3_JsonXml.PVOID;
	dintParamIndex: DINT;
	jsonMsg: Tc3_JsonXml.PVOID;
END_VAR
M_CallMethod := FALSE;
CASE intCallMethodStep OF
	0:
		IF NOT bAdsBusy AND NOT bBusy AND NOT P_bError THEN
			bBusy := TRUE;
			THIS^.M_LogMessage('Calling ADS method');
			
			// Generate JSON message
			jsonMsg := fbJson.ParseDocument('{}');
			fbJson.AddStringMember(jsonMsg, 'Target', strTargetId);			
			fbJson.AddStringMember(jsonMsg, 'Name', strMethodName);
			jsonParams := fbJson.AddObjectMember(jsonMsg, 'Params');
			FOR dintParamIndex := 1 TO GVL_DeviceAPI.uintMAX_CALL_METHOD_PARAMETERS DO
				IF LEN(arrParameters[dintParamIndex][1]) > 0 THEN
					fbJson.AddStringMember(
						jsonParams,
						arrParameters[dintParamIndex][1],
						arrParameters[dintParamIndex][2]);
				END_IF
			END_FOR
			strCommand := fbJson.GetDocument();
			
			// Set command parameters
			bSend := FALSE;
			strMessage := strCommand;
			udintGroup := udintCALL_METHOD_GROUP;
			udintOffset := udintCALL_METHOD_OFFSET;
			
			MEMSET(ADR(strResponse),0,SIZEOF(strResponse));
			// Go to next step
			intCallMethodStep := 10;
		END_IF
		
	10:
		// Wait for ADS to start running
		bSend := TRUE;
		IF bAdsBusy THEN
			intCallMethodStep := 20;
		END_IF
		
	20:
		IF NOT bAdsBusy THEN
			udintGroup := 0;
			udintOffset := 0;
			bSend := FALSE;
			IF bAdsError THEN
				THIS^.M_SetError(
					udintAdsErrorId,
					'ADS error while trying to call method!');
			ELSE
				THIS^.M_LogMessage(CONCAT('Received method response: ', strResponse));
				strReturn := strResponse;
				M_CallMethod := TRUE;
			END_IF
			bBusy := FALSE;
			intCallMethodStep := 0;
		END_IF
END_CASE
END_METHOD

(* Gets the value of a device property through an API. *)
METHOD M_GetProperty : BOOL
VAR_INPUT
	(* Name of the property to get. *)
	strPropertyName	: Tc2_System.T_MaxString;
END_VAR
VAR_OUTPUT
	(* Value of the property. *)
	strReturn	: Tc2_System.T_MaxString;
END_VAR
M_GetProperty := FALSE;
CASE intGetPropertyStep OF
	0:
		IF NOT bAdsBusy AND NOT bBusy AND NOT P_bError THEN
			bBusy := TRUE;
			THIS^.M_LogMessage('Getting property over ADS');
			
			// Set command parameters
			bSend := FALSE;
			strMessage := strPropertyName;
			udintGroup := udintGET_PROPERTY_GROUP;
			udintOffset := udintGET_PROPERTY_OFFSET;
			
			// Go to next step
			intGetPropertyStep := 10;
		END_IF
		
	10:
		// Wait for ADS to start running
		bSend := TRUE;
		IF bAdsBusy THEN
			intGetPropertyStep := 20;
		END_IF
		
	20:
		IF NOT bAdsBusy THEN
			udintGroup := 0;
			udintOffset := 0;
			bSend := FALSE;
			IF bAdsError THEN
				THIS^.M_SetError(
					udintAdsErrorId,
					'ADS error while trying to get property!');
			ELSE
				THIS^.M_LogMessage(CONCAT('Received property response: ', strResponse));
				strReturn := strResponse;
				M_GetProperty := TRUE;
			END_IF
			bBusy := FALSE;
			intGetPropertyStep := 0;
		END_IF
END_CASE
END_METHOD

(* True while a device interface command is running. *)
PROPERTY P_bDeviceInterfaceBusy : BOOL
GET
P_bDeviceInterfaceBusy := bBusy;
END_GET
END_PROPERTY

END_FUNCTION_BLOCK

// Concrete/API/FB_AdsCommandRouter
(*
Concrete implementation of a command router that works over ADS.
*)
FUNCTION_BLOCK FB_AdsCommandRouter EXTENDS FB_CommandRouter
	IMPLEMENTS I_CommandRouting
VAR_INPUT
	(* AMS Net ID of the PC that the API is running on. *)
	in_strNetId: T_AmsNetId;
	(* Port address that the API's ADS Server is running on. *)
	in_uintPort: T_AmsPort;
END_VAR
VAR_OUTPUT
END_VAR
VAR
	bRouterBusy: BOOL; // True while the router is being used by a method
	bRouteCommandBusy: BOOL; // True while M_RouteCommand is running
	fbAds: ADSRDWRTEX;
	uintRouteStep: UINT;
END_VAR
VAR CONSTANT
	udintROUTE_GROUP: UDINT := 16#1000; // Index group of the route command
	udintAWAIT_GROUP: UDINT := 16#2000; // Index group of the get result command
	udintROUTE_AND_AWAIT_GROUP: UDINT := 16#4000; // Index group of the route and return command
END_VAR

// Reset router step if route command stops being called prematurely
IF NOT bRouteCommandBusy AND uintRouteStep > 0 THEN
	uintRouteStep := 0;
	bRouterBusy := FALSE;
	THIS^.M_LogWarning('M_RouteCommand stopped being called prematurely!');
//	IF pAds > 0 THEN
//		__DELETE(pAds);
//		THIS^.M_LogWarning('Deleted ADSRDWRTEX pointer, could cause issues!');
//	END_IF
END_IF
bRouteCommandBusy := FALSE;

(* Builds the message string from input variables. *)
METHOD PRIVATE M_BuildMessage : BOOL
VAR_INPUT
	(* Unique ID of the module to call the command on. *)
	_in_strModuleId	: Tc2_System.T_MaxString;
	(* Name of the method to call. *)
	_in_strMethodName	: Tc2_System.T_MaxString;
END_VAR
VAR_IN_OUT
	(* Array of parameter key:value pairs. *)
	_inout_arrParameters : T_ApiParameterList;
END_VAR
VAR_OUTPUT
	(* Message string. *)
	_out_strMessage: T_ApiMessage;
END_VAR
VAR_INST
	_inst_fbJson: FB_JsonDynDomParser; // JSON parser function block
END_VAR
VAR
	_pJsonDoc: Tc3_JsonXml.PVOID; // Pointer to the JSON document
	_pJsonModuleId: Tc3_JsonXml.PVOID; // Pointer to the JSON module ID member
	_pJsonMethodName: Tc3_JsonXml.PVOID; // Pointer to the JSON method name member
	_pJsonParameters: Tc3_JsonXml.PVOID; // Pointer to the JSON parameters member
	_dintParamIndex: DINT; // Current parameter index
	_stParameter: ST_ApiParameter; // Current parameter being added to the JSON doc
END_VAR
// Create a blank JSON object
_pJsonDoc := _inst_fbJson.NewDocument();

// Add module ID and method name
_pJsonModuleId := _inst_fbJson.AddStringMember(_pJsonDoc, 'ModuleId', _in_strModuleId);
_pJsonMethodName := _inst_fbJson.AddStringMember(_pJsonDoc, 'MethodName', _in_strMethodName);

// Add each parameter with a key in the parameters array
_pJsonParameters := _inst_fbJson.AddObjectMember(_pJsonDoc, 'Parameters');
FOR _dintParamIndex := GVL_Api.dintPARAM_LOWER_BOUND TO GVL_Api.dintPARAM_UPPER_BOUND DO
	_stParameter := _inout_arrParameters[_dintParamIndex];
	IF LEN(_stParameter.strKey) > 0 THEN
		_inst_fbJson.AddJsonMember(_pJsonParameters, _stParameter.strKey, _stParameter.strValue);
	END_IF
END_FOR

// Output the document to strMessage
MEMSET(ADR(_out_strMessage),0,SIZEOF(_out_strMessage));
_inst_fbJson.CopyDocument(_out_strMessage, SIZEOF(_out_strMessage));

// Return true
M_BuildMessage := TRUE;
END_METHOD

METHOD PRIVATE M_ParseResult : BOOL
VAR_INPUT
	(* Result message from the API. *)
	_in_strResult: T_ApiMessage;
END_VAR
VAR_IN_OUT
	(* Any output values of the command. *)
	_inout_arrOutputs	: T_ApiParameterList;
END_VAR
VAR_OUTPUT
	(* True if the command executed without error. *)
	_out_bCommandExecuted	: BOOL;
	(* The return value of the method. *)
	_out_strReturnValue	: T_ApiParamValue;
END_VAR
VAR_INST
	_inst_fbJson: FB_JsonDynDomParser; // JSON parser function block
END_VAR
VAR
	_pJsonDoc: Tc3_JsonXml.PVOID; // Pointer to the JSON document
	_pJsonSucceeded: Tc3_JsonXml.PVOID; // Pointer to the "Successful" member
	_pJsonReturnValue: Tc3_JsonXml.PVOID; // Pointer to the "ReturnData" member
	_pJsonOutput: Tc3_JsonXml.PVOID; // Pointer to the "OutputData" member
	_pJsonIterator: Tc3_JsonXml.PVOID; // Iterator for the output data
	_pJsonIteratorEnd: Tc3_JsonXml.PVOID; // End pointer for the output data iterator
	_dintParamIndex: DINT; // Output data index
	_pOutputValue: Tc3_JsonXml.PVOID; // Pointer to the current output data value
	_strValue: T_ApiParamValue; // Output data value as a JSON string
END_VAR
// Parse the JSON string as a JSON document
_pJsonDoc := _inst_fbJson.ParseDocument(_in_strResult);

// Get success status
_pJsonSucceeded := _inst_fbJson.FindMember(_pJsonDoc, 'Successful');

// Parse the success status
IF (_pJsonSucceeded > 0) THEN
	_out_bCommandExecuted := _inst_fbJson.GetBool(_pJsonSucceeded);
	
// Throw an error if no success status member in the JSON
ELSE
	IF NOT THIS^.P_bError THEN
		THIS^.M_SetError(
			E_AdsCommandRouterError.IncorrectResponseFormat,
			'No $'Successful$' field in JSON response!');
	END_IF
END_IF

// Get return value
_pJsonReturnValue := _inst_fbJson.FindMember(_pJsonDoc, 'ReturnData');

// If there is return data, parse it
IF (_pJsonReturnValue > 0) THEN
	_inst_fbJson.CopyJson(_pJsonReturnValue, _out_strReturnValue, SIZEOF(_out_strReturnValue));
	
// Throw an error if the command executed but there is no return data
ELSIF _out_bCommandExecuted THEN
	IF NOT THIS^.P_bError THEN
		THIS^.M_SetError(
			E_AdsCommandRouterError.IncorrectResponseFormat,
			'No $'ReturnData$' field in JSON response!!');
	END_IF
END_IF

// Get output data
_pJsonOutput := _inst_fbJson.FindMember(_pJsonDoc, 'OutputData');

// If there is output data, parse it
IF (_pJsonOutput > 0) THEN
	
	// Clear output array
	FOR _dintParamIndex := GVL_Api.dintPARAM_LOWER_BOUND TO GVL_Api.dintPARAM_UPPER_BOUND DO
		_inout_arrOutputs[_dintParamIndex].strKey := '';
		MEMSET(ADR(_inout_arrOutputs[_dintParamIndex].strValue),0,SIZEOF(_inout_arrOutputs[_dintParamIndex].strValue));
	END_FOR
	
	// Initialize output data iterator and index
	_pJsonIterator := _inst_fbJson.MemberBegin(_pJsonOutput);
	_pJsonIteratorEnd := _inst_fbJson.MemberEnd(_pJsonOutput);
	_dintParamIndex := GVL_Api.dintPARAM_LOWER_BOUND;
	
	// Populate output data array with data from the JSON response data
	WHILE _pJsonIterator <> _pJsonIteratorEnd AND _dintParamIndex <= GVL_Api.dintPARAM_UPPER_BOUND DO
		// Populate the output array with the name of the current member
		_inout_arrOutputs[_dintParamIndex].strKey := _inst_fbJson.GetMemberName(_pJsonIterator);
		
		// Get the pointer to the value of the current member
		_pOutputValue := _inst_fbJson.GetMemberValue(_pJsonIterator);
		
		// Get the value as a JSON string
		_inst_fbJson.CopyJson(_pOutputValue, _strValue, SIZEOF(_strValue));
		
		// Populate the output array with the JSON string of the value
		_inout_arrOutputs[_dintParamIndex].strValue := _strValue;
		
		// Increment iterator and index
		_pJsonIterator := _inst_fbJson.NextMember(_pJsonIterator);
		_dintParamIndex := _dintParamIndex + 1;
	END_WHILE

// Throw an error if command executed but no output data member in the response JSON	
ELSIF _out_bCommandExecuted THEN
	IF NOT THIS^.P_bError THEN
		THIS^.M_SetError(
			E_AdsCommandRouterError.IncorrectResponseFormat,
			'No $'OutputData$' field in JSON response!');
	END_IF
END_IF

// Return true
M_ParseResult := TRUE;
END_METHOD

(* Routes the given command and waits for the command to finish before
returning the output data of the command. *)
METHOD M_RouteCommand : BOOL
VAR_INPUT
	(* Unique ID of the module to call the command on. *)
	_in_strModuleId	: Tc2_System.T_MaxString;
	(* Name of the method to call. *)
	_in_strMethodName : Tc2_System.T_MaxString;
	(* Timeout time for the command. *)
	_in_timeTimeout	: TIME;
END_VAR
VAR_IN_OUT
	(* Array of input parameter key:value pairs. *)
	_inout_arrParameters	: T_ApiParameterList;
	(* Array of output key:value pairs. Will be cleared and then populated with output data. *)
	_inout_arrOutputs	: T_ApiParameterList;
END_VAR
VAR_OUTPUT
	(* True if the command executed without error. Does not necessarily
	mean the command performed the task it was expected to perform, just
	means that the method returned a value. *)
	_out_bCommandExecuted	: BOOL;
	(* The return value of the method as a string. *)
	_out_strReturnValue	: T_ApiParamValue;
END_VAR
VAR_INST
	_inst_strMessage: T_ApiMessage; // JSON message that gets sent to the API
	_inst_strOutput: T_ApiMessage; // JSON message with route results received from the API
	_inst_strBuffer: T_ApiMessage; // Data buffer for ADSRDWRTEX
	_inst_bBusy: BOOL; // TRUE if the ADS function block is busy
	_inst_bErr: BOOL; // TRUE if the ADS function block has an error
	_inst_udintErrId: UDINT; // Error ID from the ADS function block if it has an error
	_inst_bWait: BOOL;
	_inst_uintStep: UINT;
END_VAR
VAR
	_udintReadCount: UDINT; // Size of the ADS read response in bytes
	_bMessageBuilt: BOOL; // Goes high once the build message method finishes
	_udintCleared: UDINT; // Number of bytes set when clearing the output string
	_bResultParsed: BOOL; // TRUE once the result parsing method finishes
	_bErrorSet: BOOL; // TRUE once an error is set on the FB
	_strBuiltMessage: T_ApiMessage; // Output of the build command method
END_VAR
VAR_INST // added by the converter: edge detectors and wires of the graphical bodies
    _w1, _w2, _w3, _w4, _w5, _w6, _w7, _w8, _w9, _w10, _w11, _w12, _w13, _w14, _w15, _w16, _w17, _w18, _w19, _w20 : BOOL;
END_VAR
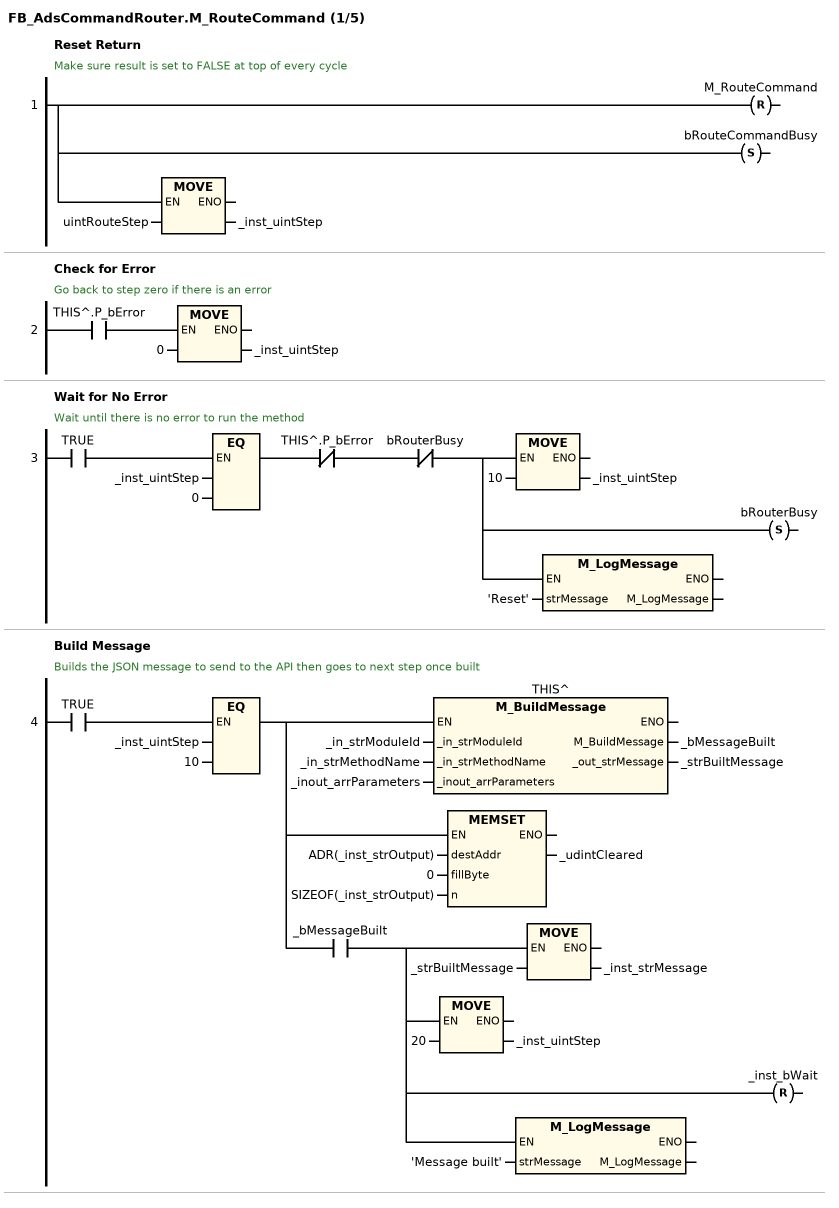
// NETWORK 1: Reset Return
// Make sure result is set to FALSE at top of every cycle
M_RouteCommand R= TRUE;
bRouteCommandBusy S= TRUE;
_inst_uintStep := uintRouteStep;

// NETWORK 2: Check for Error
// Go back to step zero if there is an error
IF THIS^.P_bError THEN _inst_uintStep := 0; END_IF

// NETWORK 3: Wait for No Error
// Wait until there is no error to run the method
_w1 := _inst_uintStep = 0 AND NOT THIS^.P_bError AND NOT bRouterBusy;
IF _w1 THEN _inst_uintStep := 10; END_IF
bRouterBusy S= _w1;
IF _w1 THEN M_LogMessage(strMessage := 'Reset'); END_IF

// NETWORK 4: Build Message
// Builds the JSON message to send to the API then goes to next step once built
_w2 := _inst_uintStep = 10;
IF _w2 THEN
    THIS^.M_BuildMessage(
        _in_strModuleId := _in_strModuleId,
        _in_strMethodName := _in_strMethodName,
        _inout_arrParameters := _inout_arrParameters,
        M_BuildMessage => _bMessageBuilt,
        _out_strMessage => _strBuiltMessage);
END_IF
IF _w2 THEN
    _udintCleared := MEMSET(destAddr := ADR(_inst_strOutput), fillByte := 0, n := SIZEOF(_inst_strOutput));
END_IF
_w3 := _w2 AND _bMessageBuilt;
IF _w3 THEN _inst_strMessage := _strBuiltMessage; END_IF
IF _w3 THEN _inst_uintStep := 20; END_IF
_inst_bWait R= _w3;
IF _w3 THEN M_LogMessage(strMessage := 'Message built'); END_IF

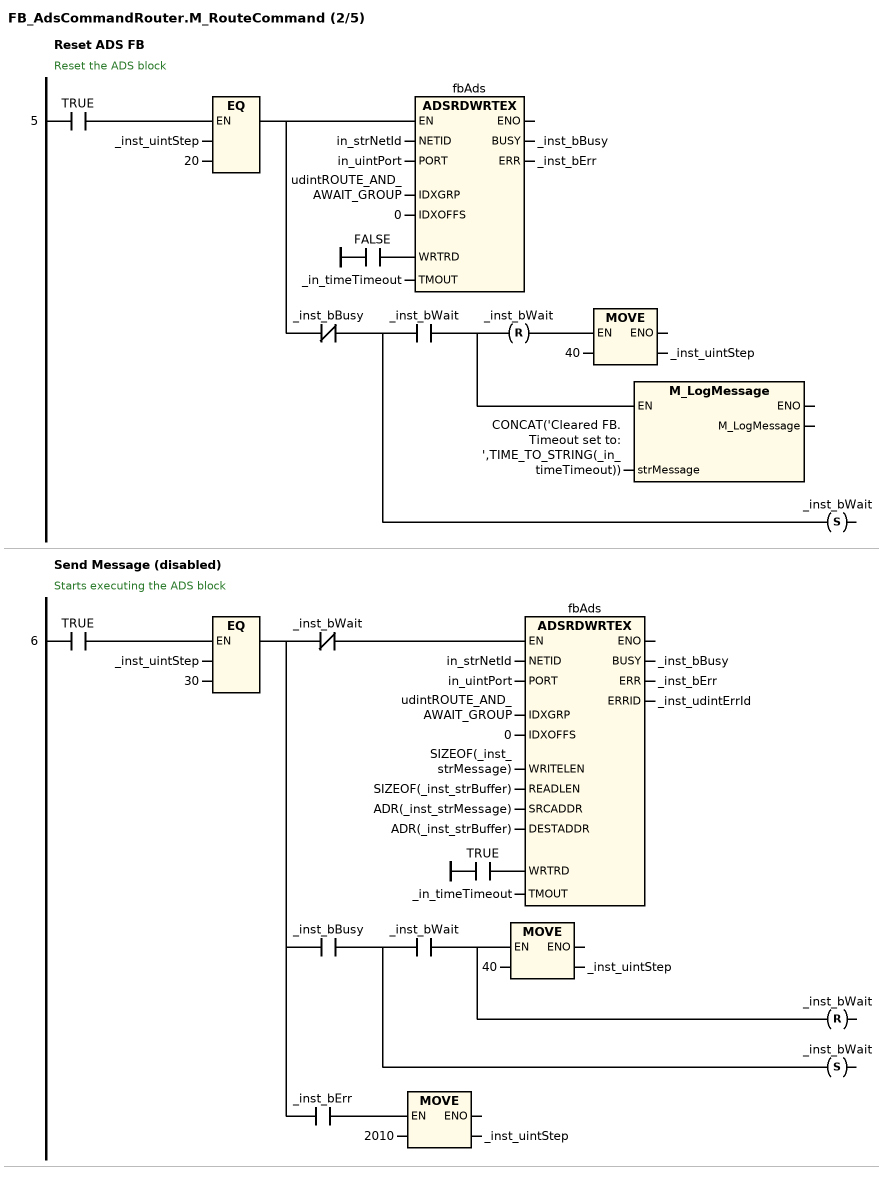
// NETWORK 5: Reset ADS FB
// Reset the ADS block
_w4 := _inst_uintStep = 20;
IF _w4 THEN
    fbAds(
        NETID := in_strNetId,
        PORT := in_uintPort,
        IDXGRP := udintROUTE_AND_AWAIT_GROUP,
        IDXOFFS := 0,
        WRTRD := FALSE,
        TMOUT := _in_timeTimeout,
        BUSY => _inst_bBusy,
        ERR => _inst_bErr); // ADSRDWRTEX
END_IF
_w5 := _w4 AND NOT _inst_bBusy;
_w6 := _w5 AND _inst_bWait;
_inst_bWait R= _w6;
IF _w6 THEN _inst_uintStep := 40; END_IF
IF _w6 THEN
    M_LogMessage(strMessage := CONCAT('Cleared FB. Timeout set to: ',TIME_TO_STRING(_in_timeTimeout)));
END_IF
_inst_bWait S= _w5;

// NETWORK 6: Send Message (disabled)
// Starts executing the ADS block
// _w7 := _inst_uintStep = 30;
// IF _w7 AND NOT _inst_bWait THEN
//     fbAds(
//         NETID := in_strNetId,
//         PORT := in_uintPort,
//         IDXGRP := udintROUTE_AND_AWAIT_GROUP,
//         IDXOFFS := 0,
//         WRITELEN := SIZEOF(_inst_strMessage),
//         READLEN := SIZEOF(_inst_strBuffer),
//         SRCADDR := ADR(_inst_strMessage),
//         DESTADDR := ADR(_inst_strBuffer),
//         WRTRD := TRUE,
//         TMOUT := _in_timeTimeout,
//         BUSY => _inst_bBusy,
//         ERR => _inst_bErr,
//         ERRID => _inst_udintErrId); // ADSRDWRTEX
// END_IF
// _w8 := _w7 AND _inst_bBusy;
// _w9 := _w8 AND _inst_bWait;
// IF _w9 THEN _inst_uintStep := 40; END_IF
// _inst_bWait R= _w9;
// _inst_bWait S= _w8;
// IF _w7 AND _inst_bErr THEN _inst_uintStep := 2010; END_IF

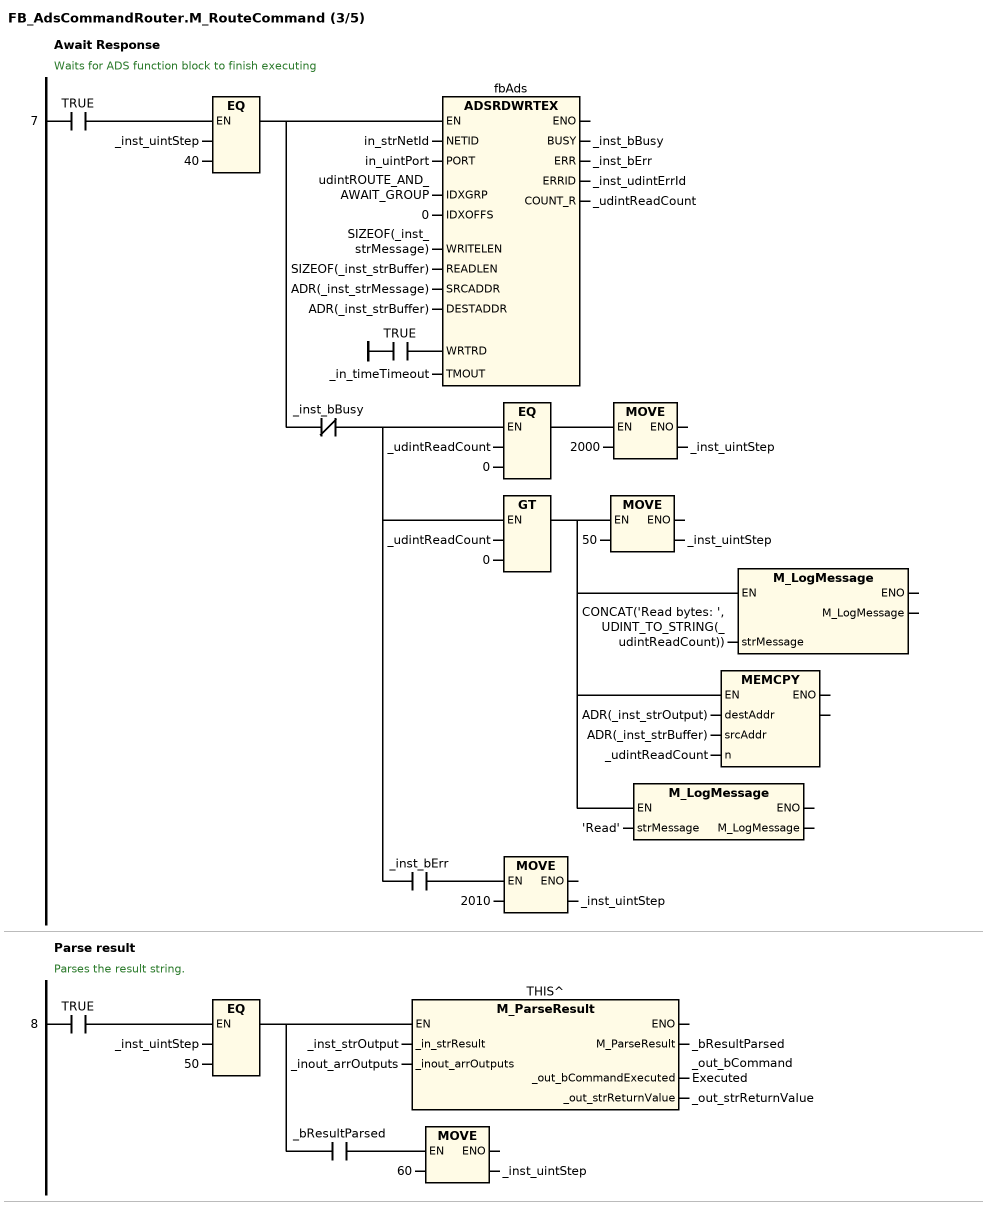
// NETWORK 7: Await Response
// Waits for ADS function block to finish executing
_w10 := _inst_uintStep = 40;
IF _w10 THEN
    fbAds(
        NETID := in_strNetId,
        PORT := in_uintPort,
        IDXGRP := udintROUTE_AND_AWAIT_GROUP,
        IDXOFFS := 0,
        WRITELEN := SIZEOF(_inst_strMessage),
        READLEN := SIZEOF(_inst_strBuffer),
        SRCADDR := ADR(_inst_strMessage),
        DESTADDR := ADR(_inst_strBuffer),
        WRTRD := TRUE,
        TMOUT := _in_timeTimeout,
        BUSY => _inst_bBusy,
        ERR => _inst_bErr,
        ERRID => _inst_udintErrId,
        COUNT_R => _udintReadCount); // ADSRDWRTEX
END_IF
_w11 := _w10 AND NOT _inst_bBusy;
IF _w11 AND _udintReadCount = 0 THEN _inst_uintStep := 2000; END_IF
_w12 := _w11 AND _udintReadCount > 0;
IF _w12 THEN _inst_uintStep := 50; END_IF
IF _w12 THEN M_LogMessage(strMessage := CONCAT('Read bytes: ', UDINT_TO_STRING(_udintReadCount))); END_IF
IF _w12 THEN
    MEMCPY(destAddr := ADR(_inst_strOutput), srcAddr := ADR(_inst_strBuffer), n := _udintReadCount);
END_IF
IF _w12 THEN M_LogMessage(strMessage := 'Read'); END_IF
IF _w11 AND _inst_bErr THEN _inst_uintStep := 2010; END_IF

// NETWORK 8: Parse result
// Parses the result string.
_w13 := _inst_uintStep = 50;
IF _w13 THEN
    THIS^.M_ParseResult(
        _in_strResult := _inst_strOutput,
        _inout_arrOutputs := _inout_arrOutputs,
        M_ParseResult => _bResultParsed,
        _out_bCommandExecuted => _out_bCommandExecuted,
        _out_strReturnValue => _out_strReturnValue);
END_IF
IF _w13 AND _bResultParsed THEN _inst_uintStep := 60; END_IF

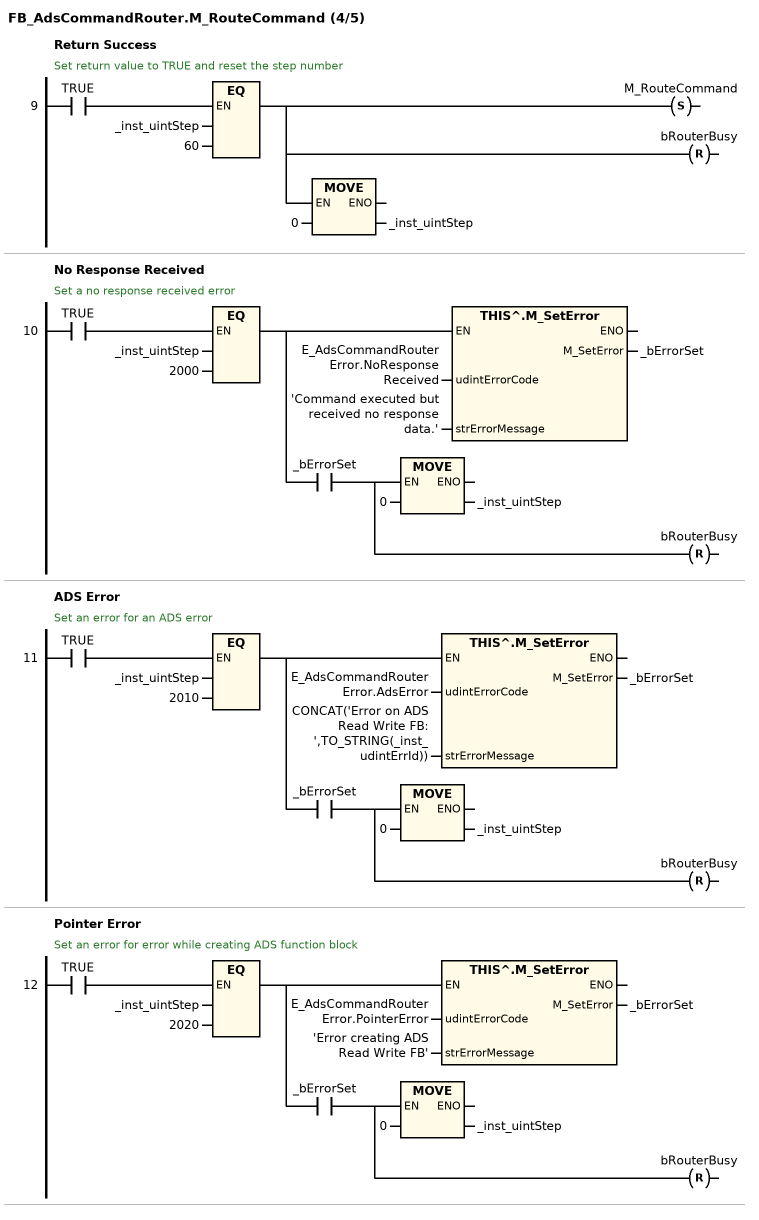
// NETWORK 9: Return Success
// Set return value to TRUE and reset the step number
_w14 := _inst_uintStep = 60;
M_RouteCommand S= _w14;
bRouterBusy R= _w14;
IF _w14 THEN _inst_uintStep := 0; END_IF

// NETWORK 10: No Response Received
// Set a no response received error
_w15 := _inst_uintStep = 2000;
IF _w15 THEN
    _bErrorSet := THIS^.M_SetError(udintErrorCode := E_AdsCommandRouterError.NoResponseReceived, strErrorMessage := 'Command executed but received no response data.');
END_IF
_w16 := _w15 AND _bErrorSet;
IF _w16 THEN _inst_uintStep := 0; END_IF
bRouterBusy R= _w16;

// NETWORK 11: ADS Error
// Set an error for an ADS error
_w17 := _inst_uintStep = 2010;
IF _w17 THEN
    _bErrorSet := THIS^.M_SetError(udintErrorCode := E_AdsCommandRouterError.AdsError, strErrorMessage := CONCAT('Error on ADS Read Write FB: ',TO_STRING(_inst_udintErrId)));
END_IF
_w18 := _w17 AND _bErrorSet;
IF _w18 THEN _inst_uintStep := 0; END_IF
bRouterBusy R= _w18;

// NETWORK 12: Pointer Error
// Set an error for error while creating ADS function block
_w19 := _inst_uintStep = 2020;
IF _w19 THEN
    _bErrorSet := THIS^.M_SetError(udintErrorCode := E_AdsCommandRouterError.PointerError, strErrorMessage := 'Error creating ADS Read Write FB');
END_IF
_w20 := _w19 AND _bErrorSet;
IF _w20 THEN _inst_uintStep := 0; END_IF
bRouterBusy R= _w20;

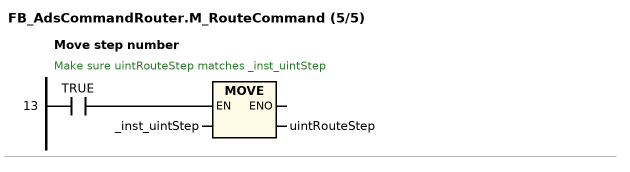
// NETWORK 13: Move step number
// Make sure uintRouteStep matches _inst_uintStep
uintRouteStep := _inst_uintStep;
END_METHOD

(* TRUE while any method in this interface is running. *)
PROPERTY P_bCommandRoutingBusy : BOOL
GET
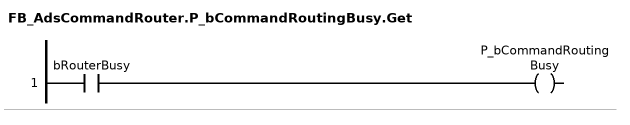
// NETWORK 1
P_bCommandRoutingBusy := bRouterBusy;
END_GET
END_PROPERTY

END_FUNCTION_BLOCK

// Concrete/API/FB_ApiDeviceTemplate
(*
	Function block for controlling a device through the Modular API.
	When making a new API device, can copy and paste this template
	and then modify accordingly.
	
	First release: June 2023 Kevin Sanita <ksanita@sensata.com>
*)
FUNCTION_BLOCK FB_ApiDeviceTemplate EXTENDS FB_Device
	IMPLEMENTS 
		I_Abortable,
		I_Connectable, 
		I_Powerable,
		I_Enableable,
		I_Resettable,
		I_Programmable
VAR_INPUT
	(* Reference to an FB_CommandRouter function block to send commands
		to a command router in the API. *)
	in_fbApi : REFERENCE TO FB_CommandRouter;
	(* ID of the API module to send router commands to. *)
	in_strApiModuleId: T_MaxString;
END_VAR
VAR_IN_OUT
END_VAR
VAR_OUTPUT
END_VAR
VAR CONSTANT
END_VAR
VAR
	bConnected: BOOL; // Value of P_bConnected
	bEnabled: BOOL; // Value of P_bEnabled
	bPoweredOn: BOOL; // Value of P_bPoweredOn
	strLoadedProgram: STRING(255); // Value of P_strLoadedProgram
	enumProgramState: E_PROGRAMSTATE; // Value of P_enumProgramState
	
	bRouterBusy: BOOL; // TRUE while M_RouterHelper is being used by a method

	bTemplateBusy: BOOL;
	bConnectBusy: BOOL;
	bDisconnectBusy: BOOL;
	bGetConnectStatusBusy: BOOL;
	bEnableBusy: BOOL;
	bDisableBusy: BOOL;
	bGetEnableStatusBusy: BOOL;
	bPowerOnBusy: BOOL;
	bPowerOffBusy: BOOL;
	bGetPowerStatusBusy: BOOL;
	bGetCurrentProgramBusy: BOOL;
	bGetProgramStateBusy: BOOL;
	bLoadProgramBusy: BOOL;
	bPauseProgramBusy: BOOL;
	bStartProgramBusy: BOOL;
	bStopProgramBusy: BOOL;
	bResetBusy: BOOL;
	bAbortBusy: BOOL;
	bRouterHelperBusy: BOOL;
	
	intTemplateStep: INT;
	intConnectStep: INT;
	intDisconnectStep: INT;
	intGetConnectStatusStep: INT;
	intEnableStep: INT;
	intDisableStep: INT;
	intGetEnableStatusStep: INT;
	intPowerOnStep: INT;
	intPowerOffStep: INT;
	intGetCurrentProgramStep: INT;
	intGetProgramStateStep: INT;
	intLoadProgramStep: INT;
	intPauseProgramStep: INT;
	intStartProgramStep: INT;
	intStopProgramStep: INT;
	intResetStep: INT;
	intAbortStep: INT;
	intGetPowerStatusStep: INT;
	intRouterHelperStep: INT;
END_VAR

A_CommandRecovery();

(* This method should establish any external connections required to use the
	functions of the device, and return TRUE and set P_bConnected to TRUE once
	connected. *)
METHOD M_Abort : BOOL
VAR CONSTANT
	_strCOMMAND_NAME : T_MaxString	:= 'Abort'; // Name of the API method
	_timeCOMMAND_TIMEOUT : TIME		:= T#30S; // Max time to receive API response
	_strSTART_MSG : T_MaxString		:= 'Aborting'; // Prints when method starts
	_strEND_MSG : T_MaxString		:= 'Aborted'; // Prints when method finishes
	_udintERROR_ID : UDINT			:= E_ApiDeviceError.FailedToAbort; // Error ID to set if command fails
	_strERROR_MSG : T_MaxString		:= 'Abort failed!'; // Error message to set if command fails
END_VAR
VAR_INST
	_inst_arrParams: T_ApiParameterList; // Parameters array
	_inst_arrOutputs: T_ApiParameterList; // Outputs array
	_inst_strRet: T_ApiParamValue; // Return string from the router
	_inst_intStep: INT; // Current method step
	_inst_fbParams: FB_ApiParamBuilder; // Parameter builder FB
END_VAR
VAR
	_bComplete: BOOL; // True if the routing finishes
	_intRet: INT; // Return string converted to an integer
	_bResult : BOOL; // Output of the method
	_pArgs: PVOID; // Arguments pointer
END_VAR
_bResult := FALSE;

// Recover from premature stop
bAbortBusy := TRUE;
_inst_intStep := intAbortStep;

// Steps
(* TEMPLATE: Parameters should be added in step 10, and output
	parsing should be added in step 30. *)
CASE _inst_intStep OF
	0: // Wait for no error and router not busy
		IF NOT THIS^.P_bError AND NOT bRouterBusy THEN
			bRouterBusy := TRUE;
			_inst_intStep := _inst_intStep + 10;
		END_IF
		
	10: // Initialize parameters
		THIS^.M_LogMessage(_strSTART_MSG);
		_inst_fbParams.M_ClearParameters();
		_pArgs := _inst_fbParams.M_AddEmptyStruct('args');
		// TEMPLATE: Add any parameters here
		_inst_fbParams.M_OutputToParameterList(_inst_arrParams);
		_inst_intStep := _inst_intStep + 10;
		
	20: // Route the command
		_bComplete := M_RouterHelper(
			_in_strMethodName := _strCOMMAND_NAME, 
			_in_timeTimeout := _timeCOMMAND_TIMEOUT,
			_inout_arrParams := _inst_arrParams,
			_inout_arrOutputs := _inst_arrOutputs,
			_out_strReturnValue=>_inst_strRet);
		
		// If route completed, move to next step
		IF _bComplete THEN
			_inst_intStep := _inst_intStep + 10;
			bRouterBusy := FALSE;
		ELSIF THIS^.P_bError THEN
			_inst_intStep := 0;
			bRouterBusy := FALSE;
		END_IF
		
	30: // Parse results
		_intRet := STRING_TO_INT(_inst_strRet);
		IF _intRet > 0 THEN
			_bResult := TRUE;
			THIS^.M_LogMessage(_strEND_MSG);
			_inst_fbParams.M_LoadFromParameterList(_inst_arrOutputs);
			// TEMPLATE: Do any parsing here
			
		// Set error if command failed
		ELSE
			THIS^.M_SetError(_udintERROR_ID, _strERROR_MSG);
		END_IF
		
		// Go back to start
		_inst_intStep := 0;
END_CASE

M_Abort := _bResult;
intAbortStep := _inst_intStep;
END_METHOD

(* This property should be TRUE while any method in this interface is actively
	executing, or FALSE otherwise. *)
PROPERTY P_bAbortBusy : BOOL
GET
P_bAbortBusy := bRouterBusy;
END_GET
END_PROPERTY

(* This method should establish any external connections required to use the
	functions of the device, and return TRUE and set P_bConnected to TRUE once
	connected. *)
METHOD M_Connect : BOOL
VAR CONSTANT
	_strCOMMAND_NAME : T_MaxString	:= 'Connect'; // Name of the API method
	_timeCOMMAND_TIMEOUT : TIME		:= T#30S; // Max time to receive API response
	_strSTART_MSG : T_MaxString		:= 'Connecting'; // Prints when method starts
	_strEND_MSG : T_MaxString		:= 'Connected'; // Prints when method finishes
	_udintERROR_ID : UDINT			:= E_ApiDeviceError.FailedToConnect; // Error ID to set if command fails
	_strERROR_MSG : T_MaxString		:= 'Failed to connect!'; // Error message to set if command fails
END_VAR
VAR_INST
	_inst_arrParams: T_ApiParameterList; // Parameters array
	_inst_arrOutputs: T_ApiParameterList; // Outputs array
	_inst_strRet: T_ApiParamValue; // Return string from the router
	_inst_intStep: INT; // Current method step
	_inst_fbParams: FB_ApiParamBuilder; // Parameter builder FB
END_VAR
VAR
	_bComplete: BOOL; // True if the routing finishes
	_intRet: INT; // Return string converted to an integer
	_bResult : BOOL; // Output of the method
	_pArgs: PVOID; // Arguments pointer
END_VAR
_bResult := FALSE;

// Recover from premature stop
bConnectBusy := TRUE;
_inst_intStep := intConnectStep;

// Steps
(* TEMPLATE: Parameters should be added in step 10, and output
	parsing should be added in step 30. *)
CASE _inst_intStep OF
	0: // Wait for no error and router not busy
		IF NOT THIS^.P_bError AND NOT bRouterBusy THEN
			bRouterBusy := TRUE;
			_inst_intStep := _inst_intStep + 10;
		END_IF
		
	10: // Initialize parameters
		THIS^.M_LogMessage(_strSTART_MSG);
		_inst_fbParams.M_ClearParameters();
		_pArgs := _inst_fbParams.M_AddEmptyStruct('args');
		// TEMPLATE: Add any parameters here
		_inst_fbParams.M_OutputToParameterList(_inst_arrParams);
		_inst_intStep := _inst_intStep + 10;
		
	20: // Route the command
		_bComplete := M_RouterHelper(
			_in_strMethodName := _strCOMMAND_NAME, 
			_in_timeTimeout := _timeCOMMAND_TIMEOUT,
			_inout_arrParams := _inst_arrParams,
			_inout_arrOutputs := _inst_arrOutputs,
			_out_strReturnValue=>_inst_strRet);
		
		// If route completed, move to next step
		IF _bComplete THEN
			_inst_intStep := _inst_intStep + 10;
			bRouterBusy := FALSE;
		ELSIF THIS^.P_bError THEN
			_inst_intStep := 0;
			bRouterBusy := FALSE;
		END_IF
		
	30: // Parse results
		_intRet := STRING_TO_INT(_inst_strRet);
		IF _intRet > 0 THEN
			_bResult := TRUE;
			THIS^.M_LogMessage(_strEND_MSG);
			_inst_fbParams.M_LoadFromParameterList(_inst_arrOutputs);
			// TEMPLATE: Do any parsing here
			bConnected := TRUE;
			
		// Set error if command failed
		ELSE
			THIS^.M_SetError(_udintERROR_ID, _strERROR_MSG);
		END_IF
		
		// Go back to start
		_inst_intStep := 0;
END_CASE

M_Connect := _bResult;
intConnectStep := _inst_intStep;
END_METHOD

(* This method should break any connections established by M_Connect. It should
	immediately set P_bConnected to false unless all connections are known to
	be still active, and return TRUE once those connections are all fully
	disconnected. *)
METHOD M_Disconnect : BOOL
VAR CONSTANT
	_strCOMMAND_NAME : T_MaxString	:= 'Disconnect'; // Name of the API method
	_timeCOMMAND_TIMEOUT : TIME		:= T#30S; // Max time to receive API response
	_strSTART_MSG : T_MaxString		:= 'Disconnecting'; // Prints when method starts
	_strEND_MSG : T_MaxString		:= 'Disconnected'; // Prints when method finishes
	_udintERROR_ID : UDINT			:= E_ApiDeviceError.FailedToDisconnect; // Error ID to set if command fails
	_strERROR_MSG : T_MaxString		:= 'Failed to disconnect!'; // Error message to set if command fails
END_VAR
VAR_INST
	_inst_arrParams: T_ApiParameterList; // Parameters array
	_inst_arrOutputs: T_ApiParameterList; // Outputs array
	_inst_strRet: T_ApiParamValue; // Return string from the router
	_inst_intStep: INT; // Current method step
	_inst_fbParams: FB_ApiParamBuilder; // Parameter builder FB
END_VAR
VAR
	_bComplete: BOOL; // True if the routing finishes
	_intRet: INT; // Return string converted to an integer
	_bResult : BOOL; // Output of the method
	_pArgs: PVOID; // Arguments pointer
END_VAR
_bResult := FALSE;

// Recover from premature stop
bDisconnectBusy := TRUE;
_inst_intStep := intDisconnectStep;

// Steps
(* TEMPLATE: Parameters should be added in step 10, and output
	parsing should be added in step 30. *)
CASE _inst_intStep OF
	0: // Wait for no error and router not busy
		IF NOT THIS^.P_bError AND NOT bRouterBusy THEN
			bRouterBusy := TRUE;
			_inst_intStep := _inst_intStep + 10;
		END_IF
		
	10: // Initialize parameters
		THIS^.M_LogMessage(_strSTART_MSG);
		_inst_fbParams.M_ClearParameters();
		_pArgs := _inst_fbParams.M_AddEmptyStruct('args');
		// TEMPLATE: Add any parameters here
		_inst_fbParams.M_OutputToParameterList(_inst_arrParams);
		_inst_intStep := _inst_intStep + 10;
		
	20: // Route the command
		_bComplete := M_RouterHelper(
			_in_strMethodName := _strCOMMAND_NAME, 
			_in_timeTimeout := _timeCOMMAND_TIMEOUT,
			_inout_arrParams := _inst_arrParams,
			_inout_arrOutputs := _inst_arrOutputs,
			_out_strReturnValue=>_inst_strRet);
		
		// If route completed, move to next step
		IF _bComplete THEN
			_inst_intStep := _inst_intStep + 10;
			bRouterBusy := FALSE;
		ELSIF THIS^.P_bError THEN
			_inst_intStep := 0;
			bRouterBusy := FALSE;
		END_IF
		
	30: // Parse results
		_intRet := STRING_TO_INT(_inst_strRet);
		IF _intRet > 0 THEN
			_bResult := TRUE;
			THIS^.M_LogMessage(_strEND_MSG);
			_inst_fbParams.M_LoadFromParameterList(_inst_arrOutputs);
			// TEMPLATE: Do any parsing here
			bConnected := FALSE;
			
		// Set error if command failed
		ELSE
			THIS^.M_SetError(_udintERROR_ID, _strERROR_MSG);
		END_IF
		
		// Go back to start
		_inst_intStep := 0;
END_CASE

M_Disconnect := _bResult;
intDisconnectStep := _inst_intStep;
END_METHOD

(* This method should explicitly check the connection status of the device.
	Once the connection status is known, this method should return TRUE.
	If this method fails, P_bConnected should be set to FALSE since the device
	is not absolutely known to still be connected. *)
METHOD M_GetConnectStatus : BOOL
VAR_OUTPUT
	(* This should return TRUE if all connections required to make the device
		function properly are known to be connected, and FALSE otherwise. *)
	bConnected	: BOOL;
END_VAR
VAR CONSTANT
	_strCOMMAND_NAME : T_MaxString	:= 'GetConnectStatus'; // Name of the API method
	_timeCOMMAND_TIMEOUT : TIME		:= T#5S; // Max time to receive API response
	_strSTART_MSG : T_MaxString		:= 'Getting connection status'; // Prints when method starts
	_strEND_MSG : T_MaxString		:= 'Received connection status'; // Prints when method finishes
	_udintERROR_ID : UDINT			:= E_ApiDeviceError.FailedToGetConnectStatus; // Error ID to set if command fails
	_strERROR_MSG : T_MaxString		:= 'Failed to get connection status!'; // Error message to set if command fails
END_VAR
VAR_INST
	_inst_arrParams: T_ApiParameterList; // Parameters array
	_inst_arrOutputs: T_ApiParameterList; // Outputs array
	_inst_strRet: T_ApiParamValue; // Return string from the router
	_inst_intStep: INT; // Current method step
	_inst_fbParams: FB_ApiParamBuilder; // Parameter builder FB
END_VAR
VAR
	_bComplete: BOOL; // True if the routing finishes
	_intRet: INT; // Return string converted to an integer
	_bResult : BOOL; // Output of the method
	_pArgs: PVOID; // Arguments pointer
END_VAR
_bResult := FALSE;

// Recover from premature stop
bGetConnectStatusBusy := TRUE;
_inst_intStep := intGetConnectStatusStep;

// Steps
(* TEMPLATE: Parameters should be added in step 10, and output
	parsing should be added in step 30. *)
CASE _inst_intStep OF
	0: // Wait for no error and router not busy
		IF NOT THIS^.P_bError AND NOT bRouterBusy THEN
			bRouterBusy := TRUE;
			_inst_intStep := _inst_intStep + 10;
		END_IF
		
	10: // Initialize parameters
		THIS^.M_LogMessage(_strSTART_MSG);
		_inst_fbParams.M_ClearParameters();
		_pArgs := _inst_fbParams.M_AddEmptyStruct('args');
		// TEMPLATE: Add any parameters here
		_inst_fbParams.M_OutputToParameterList(_inst_arrParams);
		_inst_intStep := _inst_intStep + 10;
		
	20: // Route the command
		_bComplete := M_RouterHelper(
			_in_strMethodName := _strCOMMAND_NAME, 
			_in_timeTimeout := _timeCOMMAND_TIMEOUT,
			_inout_arrParams := _inst_arrParams,
			_inout_arrOutputs := _inst_arrOutputs,
			_out_strReturnValue=>_inst_strRet);
		
		// If route completed, move to next step
		IF _bComplete THEN
			_inst_intStep := _inst_intStep + 10;
			bRouterBusy := FALSE;
		ELSIF THIS^.P_bError THEN
			_inst_intStep := 0;
			bRouterBusy := FALSE;
		END_IF
		
	30: // Parse results
		_intRet := STRING_TO_INT(_inst_strRet);
		IF _intRet > 0 THEN
			_bResult := TRUE;
			THIS^.M_LogMessage(_strEND_MSG);
			_inst_fbParams.M_LoadFromParameterList(_inst_arrOutputs);
			// TEMPLATE: Do any parsing here
			THIS^.bConnected := _inst_fbParams.M_ParseBool(
				_inst_fbParams.M_GetParameter('connected'));
			bConnected := THIS^.bConnected;
			
		// Set error if command failed
		ELSE
			THIS^.M_SetError(_udintERROR_ID, _strERROR_MSG);
		END_IF
		
		// Go back to start
		_inst_intStep := 0;
END_CASE

M_GetConnectStatus := _bResult;
intGetConnectStatusStep := _inst_intStep;
END_METHOD

(* This property should be TRUE while any method in this interface is actively
	executing, or FALSE otherwise. *)
PROPERTY P_bConnectBusy : BOOL
GET
P_bConnectBusy := bRouterBusy;
END_GET
END_PROPERTY

(* This should be set to TRUE if M_Connect is successful or M_GetConnectStatus
	determines the device to be connected, and set to FALSE if M_Disconnect is
	called at all, M_GetConnectStatus fails, or M_GetConnectStatus determines
	the device to be not connected. *)
PROPERTY P_bConnected : BOOL
GET
P_bConnected := bConnected;
END_GET
END_PROPERTY

(* This method should return to the device to the state it was prior to being
	enabled. P_bEnabled should be immediately set to false unless the status of
	the device is explicitly known to still be enabled. After being disabled,
	the device should typically be unable to perform process steps. Once
	successfully disabled, this method should return TRUE. *)
METHOD M_Disable : BOOL
VAR CONSTANT
	_strCOMMAND_NAME : T_MaxString	:= 'Disable'; // Name of the API method
	_timeCOMMAND_TIMEOUT : TIME		:= T#30S; // Max time to receive API response
	_strSTART_MSG : T_MaxString		:= 'Disabling'; // Prints when method starts
	_strEND_MSG : T_MaxString		:= 'Disabled'; // Prints when method finishes
	_udintERROR_ID : UDINT			:= E_ApiDeviceError.FailedToDisable; // Error ID to set if command fails
	_strERROR_MSG : T_MaxString		:= 'Failed to disable!'; // Error message to set if command fails
END_VAR
VAR_INST
	_inst_arrParams: T_ApiParameterList; // Parameters array
	_inst_arrOutputs: T_ApiParameterList; // Outputs array
	_inst_strRet: T_ApiParamValue; // Return string from the router
	_inst_intStep: INT; // Current method step
	_inst_fbParams: FB_ApiParamBuilder; // Parameter builder FB
END_VAR
VAR
	_bComplete: BOOL; // True if the routing finishes
	_intRet: INT; // Return string converted to an integer
	_bResult : BOOL; // Output of the method
	_pArgs: PVOID; // Arguments pointer
END_VAR
_bResult := FALSE;

// Recover from premature stop
bDisableBusy := TRUE;
_inst_intStep := intDisableStep;

// Steps
(* TEMPLATE: Parameters should be added in step 10, and output
	parsing should be added in step 30. *)
CASE _inst_intStep OF
	0: // Wait for no error and router not busy
		IF NOT THIS^.P_bError AND NOT bRouterBusy THEN
			bRouterBusy := TRUE;
			_inst_intStep := _inst_intStep + 10;
		END_IF
		
	10: // Initialize parameters
		THIS^.M_LogMessage(_strSTART_MSG);
		_inst_fbParams.M_ClearParameters();
		_pArgs := _inst_fbParams.M_AddEmptyStruct('args');
		// TEMPLATE: Add any parameters here
		_inst_fbParams.M_OutputToParameterList(_inst_arrParams);
		_inst_intStep := _inst_intStep + 10;
		
	20: // Route the command
		_bComplete := M_RouterHelper(
			_in_strMethodName := _strCOMMAND_NAME, 
			_in_timeTimeout := _timeCOMMAND_TIMEOUT,
			_inout_arrParams := _inst_arrParams,
			_inout_arrOutputs := _inst_arrOutputs,
			_out_strReturnValue=>_inst_strRet);
		
		// If route completed, move to next step
		IF _bComplete THEN
			_inst_intStep := _inst_intStep + 10;
			bRouterBusy := FALSE;
		ELSIF THIS^.P_bError THEN
			_inst_intStep := 0;
			bRouterBusy := FALSE;
		END_IF
		
	30: // Parse results
		_intRet := STRING_TO_INT(_inst_strRet);
		IF _intRet > 0 THEN
			_bResult := TRUE;
			THIS^.M_LogMessage(_strEND_MSG);
			_inst_fbParams.M_LoadFromParameterList(_inst_arrOutputs);
			// TEMPLATE: Do any parsing here
			bEnabled := FALSE;
			
		// Set error if command failed
		ELSE
			THIS^.M_SetError(_udintERROR_ID, _strERROR_MSG);
		END_IF
		
		// Go back to start
		_inst_intStep := 0;
END_CASE

M_Disable := _bResult;
intDisableStep := _inst_intStep;
END_METHOD

(* This method should perform any tasks that must be performed after a device
	is energized, but prior to the device being used in a process, and then
	return TRUE and set P_bEnabled to TRUE once those tasks are completed. *)
METHOD M_Enable : BOOL
VAR CONSTANT
	_strCOMMAND_NAME : T_MaxString	:= 'Enable'; // Name of the API method
	_timeCOMMAND_TIMEOUT : TIME		:= T#30S; // Max time to receive API response
	_strSTART_MSG : T_MaxString		:= 'Enabling'; // Prints when method starts
	_strEND_MSG : T_MaxString		:= 'Enabled'; // Prints when method finishes
	_udintERROR_ID : UDINT			:= E_ApiDeviceError.FailedToEnable; // Error ID to set if command fails
	_strERROR_MSG : T_MaxString		:= 'Failed to enable!'; // Error message to set if command fails
END_VAR
VAR_INST
	_inst_arrParams: T_ApiParameterList; // Parameters array
	_inst_arrOutputs: T_ApiParameterList; // Outputs array
	_inst_strRet: T_ApiParamValue; // Return string from the router
	_inst_intStep: INT; // Current method step
	_inst_fbParams: FB_ApiParamBuilder; // Parameter builder FB
END_VAR
VAR
	_bComplete: BOOL; // True if the routing finishes
	_intRet: INT; // Return string converted to an integer
	_bResult : BOOL; // Output of the method
	_pArgs: PVOID; // Arguments pointer
END_VAR
_bResult := FALSE;

// Recover from premature stop
bEnableBusy := TRUE;
_inst_intStep := intEnableStep;

// Steps
(* TEMPLATE: Parameters should be added in step 10, and output
	parsing should be added in step 30. *)
CASE _inst_intStep OF
	0: // Wait for no error and router not busy
		IF NOT THIS^.P_bError AND NOT bRouterBusy THEN
			bRouterBusy := TRUE;
			_inst_intStep := _inst_intStep + 10;
		END_IF
		
	10: // Initialize parameters
		THIS^.M_LogMessage(_strSTART_MSG);
		_inst_fbParams.M_ClearParameters();
		_pArgs := _inst_fbParams.M_AddEmptyStruct('args');
		// TEMPLATE: Add any parameters here
		_inst_fbParams.M_OutputToParameterList(_inst_arrParams);
		_inst_intStep := _inst_intStep + 10;
		
	20: // Route the command
		_bComplete := M_RouterHelper(
			_in_strMethodName := _strCOMMAND_NAME, 
			_in_timeTimeout := _timeCOMMAND_TIMEOUT,
			_inout_arrParams := _inst_arrParams,
			_inout_arrOutputs := _inst_arrOutputs,
			_out_strReturnValue=>_inst_strRet);
		
		// If route completed, move to next step
		IF _bComplete THEN
			_inst_intStep := _inst_intStep + 10;
			bRouterBusy := FALSE;
		ELSIF THIS^.P_bError THEN
			_inst_intStep := 0;
			bRouterBusy := FALSE;
		END_IF
		
	30: // Parse results
		_intRet := STRING_TO_INT(_inst_strRet);
		IF _intRet > 0 THEN
			_bResult := TRUE;
			THIS^.M_LogMessage(_strEND_MSG);
			_inst_fbParams.M_LoadFromParameterList(_inst_arrOutputs);
			// TEMPLATE: Do any parsing here
			bEnabled := TRUE;
			
		// Set error if command failed
		ELSE
			THIS^.M_SetError(_udintERROR_ID, _strERROR_MSG);
		END_IF
		
		// Go back to start
		_inst_intStep := 0;
END_CASE

M_Enable := _bResult;
intEnableStep := _inst_intStep;
END_METHOD

(* This method should explicitly check the enable status of the device.
	Once the enable status is known, this method should return TRUE.
	If this method fails, P_bEnabled should be set to FALSE since the device
	is not absolutely known to still be enabled. *)
METHOD M_GetEnableStatus : BOOL
VAR_OUTPUT
	(* This should return TRUE if the device is explicitly known to be
		enabled, or FALSE otherwise. *)
	bEnabled	: BOOL;
END_VAR
VAR CONSTANT
	_strCOMMAND_NAME : T_MaxString	:= 'GetEnableStatus'; // Name of the API method
	_timeCOMMAND_TIMEOUT : TIME		:= T#5S; // Max time to receive API response
	_strSTART_MSG : T_MaxString		:= 'Getting enable status'; // Prints when method starts
	_strEND_MSG : T_MaxString		:= 'Received enable status'; // Prints when method finishes
	_udintERROR_ID : UDINT			:= E_ApiDeviceError.FailedToGetEnableStatus; // Error ID to set if command fails
	_strERROR_MSG : T_MaxString		:= 'Failed to get enable status!'; // Error message to set if command fails
END_VAR
VAR_INST
	_inst_arrParams: T_ApiParameterList; // Parameters array
	_inst_arrOutputs: T_ApiParameterList; // Outputs array
	_inst_strRet: T_ApiParamValue; // Return string from the router
	_inst_intStep: INT; // Current method step
	_inst_fbParams: FB_ApiParamBuilder; // Parameter builder FB
END_VAR
VAR
	_bComplete: BOOL; // True if the routing finishes
	_intRet: INT; // Return string converted to an integer
	_bResult : BOOL; // Output of the method
	_pArgs: PVOID; // Arguments pointer
END_VAR
_bResult := FALSE;

// Recover from premature stop
bGetEnableStatusBusy := TRUE;
_inst_intStep := intGetEnableStatusStep;

// Steps
(* TEMPLATE: Parameters should be added in step 10, and output
	parsing should be added in step 30. *)
CASE _inst_intStep OF
	0: // Wait for no error and router not busy
		IF NOT THIS^.P_bError AND NOT bRouterBusy THEN
			bRouterBusy := TRUE;
			_inst_intStep := _inst_intStep + 10;
		END_IF
		
	10: // Initialize parameters
		THIS^.M_LogMessage(_strSTART_MSG);
		_inst_fbParams.M_ClearParameters();
		_pArgs := _inst_fbParams.M_AddEmptyStruct('args');
		// TEMPLATE: Add any parameters here
		_inst_fbParams.M_OutputToParameterList(_inst_arrParams);
		_inst_intStep := _inst_intStep + 10;
		
	20: // Route the command
		_bComplete := M_RouterHelper(
			_in_strMethodName := _strCOMMAND_NAME, 
			_in_timeTimeout := _timeCOMMAND_TIMEOUT,
			_inout_arrParams := _inst_arrParams,
			_inout_arrOutputs := _inst_arrOutputs,
			_out_strReturnValue=>_inst_strRet);
		
		// If route completed, move to next step
		IF _bComplete THEN
			_inst_intStep := _inst_intStep + 10;
			bRouterBusy := FALSE;
		ELSIF THIS^.P_bError THEN
			_inst_intStep := 0;
			bRouterBusy := FALSE;
		END_IF
		
	30: // Parse results
		_intRet := STRING_TO_INT(_inst_strRet);
		IF _intRet > 0 THEN
			_bResult := TRUE;
			THIS^.M_LogMessage(_strEND_MSG);
			_inst_fbParams.M_LoadFromParameterList(_inst_arrOutputs);
			// TEMPLATE: Do any parsing here
			THIS^.bEnabled := _inst_fbParams.M_ParseBool(
				_inst_fbParams.M_GetParameter('enabled'));
			bEnabled := THIS^.bEnabled;
			
		// Set error if command failed
		ELSE
			THIS^.M_SetError(_udintERROR_ID, _strERROR_MSG);
		END_IF
		
		// Go back to start
		_inst_intStep := 0;
END_CASE

M_GetEnableStatus := _bResult;
intGetEnableStatusStep := _inst_intStep;
END_METHOD

(* This property should be TRUE while any method in this interface is actively
	executing, or FALSE otherwise. *)
PROPERTY P_bEnableBusy : BOOL
GET
P_bEnableBusy := bRouterBusy;
END_GET
END_PROPERTY

(* This should be set to TRUE if M_Enable is successful or M_GetEnableStatus
	determines the device to be enabled, and set to FALSE if M_Disable is
	called at all, M_GetEnableStatus fails, or M_GetEnableStatus determines
	the device to be not enabled. *)
PROPERTY P_bEnabled : BOOL
GET
P_bEnabled := bEnabled;
END_GET
END_PROPERTY

(* This method should explicitly check the power status of the device.
	Once the power status is known, this method should return TRUE.
	If this method fails, P_bPoweredOn should be set to FALSE since the device
	is not absolutely known to still be powered on. *)
METHOD M_GetPowerStatus : BOOL
VAR_OUTPUT
	(* This should return TRUE if the device is explicitly known to be
		powered on, or FALSE otherwise. *)
	bPoweredOn	: BOOL;
END_VAR
VAR CONSTANT
	_strCOMMAND_NAME : T_MaxString	:= 'GetPowerStatus'; // Name of the API method
	_timeCOMMAND_TIMEOUT : TIME		:= T#5S; // Max time to receive API response
	_strSTART_MSG : T_MaxString		:= 'Getting power status'; // Prints when method starts
	_strEND_MSG : T_MaxString		:= 'Received power status'; // Prints when method finishes
	_udintERROR_ID : UDINT			:= E_ApiDeviceError.FailedToGetPowerStatus; // Error ID to set if command fails
	_strERROR_MSG : T_MaxString		:= 'Failed to get power status!'; // Error message to set if command fails
END_VAR
VAR_INST
	_inst_arrParams: T_ApiParameterList; // Parameters array
	_inst_arrOutputs: T_ApiParameterList; // Outputs array
	_inst_strRet: T_ApiParamValue; // Return string from the router
	_inst_intStep: INT; // Current method step
	_inst_fbParams: FB_ApiParamBuilder; // Parameter builder FB
END_VAR
VAR
	_bComplete: BOOL; // True if the routing finishes
	_intRet: INT; // Return string converted to an integer
	_bResult : BOOL; // Output of the method
	_pArgs: PVOID; // Arguments pointer
END_VAR
_bResult := FALSE;

// Recover from premature stop
bGetPowerStatusBusy := TRUE;
_inst_intStep := intGetPowerStatusStep;

// Steps
(* TEMPLATE: Parameters should be added in step 10, and output
	parsing should be added in step 30. *)
CASE _inst_intStep OF
	0: // Wait for no error and router not busy
		IF NOT THIS^.P_bError AND NOT bRouterBusy THEN
			bRouterBusy := TRUE;
			_inst_intStep := _inst_intStep + 10;
		END_IF
		
	10: // Initialize parameters
		THIS^.M_LogMessage(_strSTART_MSG);
		_inst_fbParams.M_ClearParameters();
		_pArgs := _inst_fbParams.M_AddEmptyStruct('args');
		// TEMPLATE: Add any parameters here
		_inst_fbParams.M_OutputToParameterList(_inst_arrParams);
		_inst_intStep := _inst_intStep + 10;
		
	20: // Route the command
		_bComplete := M_RouterHelper(
			_in_strMethodName := _strCOMMAND_NAME, 
			_in_timeTimeout := _timeCOMMAND_TIMEOUT,
			_inout_arrParams := _inst_arrParams,
			_inout_arrOutputs := _inst_arrOutputs,
			_out_strReturnValue=>_inst_strRet);
		
		// If route completed, move to next step
		IF _bComplete THEN
			_inst_intStep := _inst_intStep + 10;
			bRouterBusy := FALSE;
		ELSIF THIS^.P_bError THEN
			_inst_intStep := 0;
			bRouterBusy := FALSE;
		END_IF
		
	30: // Parse results
		_intRet := STRING_TO_INT(_inst_strRet);
		IF _intRet > 0 THEN
			_bResult := TRUE;
			THIS^.M_LogMessage(_strEND_MSG);
			_inst_fbParams.M_LoadFromParameterList(_inst_arrOutputs);
			// TEMPLATE: Do any parsing here
			THIS^.bPoweredOn := _inst_fbParams.M_ParseBool(
				_inst_fbParams.M_GetParameter('poweredOn'));
			bPoweredOn := THIS^.bPoweredOn;
			
		// Set error if command failed
		ELSE
			THIS^.M_SetError(_udintERROR_ID, _strERROR_MSG);
		END_IF
		
		// Go back to start
		_inst_intStep := 0;
END_CASE

M_GetPowerStatus := _bResult;
intGetPowerStatusStep := _inst_intStep;
END_METHOD

(* This method should de-energize the device and then return TRUE once
	successful. P_bPoweredOn should be set to FALSE immediately when this is
	called unless the device is explicitly known to still be powered on. *)
METHOD M_PowerOff : BOOL
VAR CONSTANT
	_strCOMMAND_NAME : T_MaxString	:= 'PowerOff'; // Name of the API method
	_timeCOMMAND_TIMEOUT : TIME		:= T#30S; // Max time to receive API response
	_strSTART_MSG : T_MaxString		:= 'Powering off'; // Prints when method starts
	_strEND_MSG : T_MaxString		:= 'Powered off'; // Prints when method finishes
	_udintERROR_ID : UDINT			:= E_ApiDeviceError.FailedToPowerOff; // Error ID to set if command fails
	_strERROR_MSG : T_MaxString		:= 'Failed to power off!'; // Error message to set if command fails
END_VAR
VAR_INST
	_inst_arrParams: T_ApiParameterList; // Parameters array
	_inst_arrOutputs: T_ApiParameterList; // Outputs array
	_inst_strRet: T_ApiParamValue; // Return string from the router
	_inst_intStep: INT; // Current method step
	_inst_fbParams: FB_ApiParamBuilder; // Parameter builder FB
END_VAR
VAR
	_bComplete: BOOL; // True if the routing finishes
	_intRet: INT; // Return string converted to an integer
	_bResult : BOOL; // Output of the method
	_pArgs: PVOID; // Arguments pointer
END_VAR
_bResult := FALSE;

// Recover from premature stop
bPowerOffBusy := TRUE;
_inst_intStep := intPowerOffStep;

// Steps
(* TEMPLATE: Parameters should be added in step 10, and output
	parsing should be added in step 30. *)
CASE _inst_intStep OF
	0: // Wait for no error and router not busy
		IF NOT THIS^.P_bError AND NOT bRouterBusy THEN
			bRouterBusy := TRUE;
			_inst_intStep := _inst_intStep + 10;
		END_IF
		
	10: // Initialize parameters
		THIS^.M_LogMessage(_strSTART_MSG);
		_inst_fbParams.M_ClearParameters();
		_pArgs := _inst_fbParams.M_AddEmptyStruct('args');
		// TEMPLATE: Add any parameters here
		_inst_fbParams.M_OutputToParameterList(_inst_arrParams);
		_inst_intStep := _inst_intStep + 10;
		
	20: // Route the command
		_bComplete := M_RouterHelper(
			_in_strMethodName := _strCOMMAND_NAME, 
			_in_timeTimeout := _timeCOMMAND_TIMEOUT,
			_inout_arrParams := _inst_arrParams,
			_inout_arrOutputs := _inst_arrOutputs,
			_out_strReturnValue=>_inst_strRet);
		
		// If route completed, move to next step
		IF _bComplete THEN
			_inst_intStep := _inst_intStep + 10;
			bRouterBusy := FALSE;
		ELSIF THIS^.P_bError THEN
			_inst_intStep := 0;
			bRouterBusy := FALSE;
		END_IF
		
	30: // Parse results
		_intRet := STRING_TO_INT(_inst_strRet);
		IF _intRet > 0 THEN
			_bResult := TRUE;
			THIS^.M_LogMessage(_strEND_MSG);
			_inst_fbParams.M_LoadFromParameterList(_inst_arrOutputs);
			// TEMPLATE: Do any parsing here
			bPoweredOn := FALSE;
			
		// Set error if command failed
		ELSE
			THIS^.M_SetError(_udintERROR_ID, _strERROR_MSG);
		END_IF
		
		// Go back to start
		_inst_intStep := 0;
END_CASE

M_PowerOff := _bResult;
intPowerOffStep := _inst_intStep;
END_METHOD

(* This method should energize the device and then return TRUE and set
	P_bPoweredOn to TRUE once successful. *)
METHOD M_PowerOn : BOOL
VAR CONSTANT
	_strCOMMAND_NAME : T_MaxString	:= 'PowerOn'; // Name of the API method
	_timeCOMMAND_TIMEOUT : TIME		:= T#30S; // Max time to receive API response
	_strSTART_MSG : T_MaxString		:= 'Powering on'; // Prints when method starts
	_strEND_MSG : T_MaxString		:= 'Powered on'; // Prints when method finishes
	_udintERROR_ID : UDINT			:= E_ApiDeviceError.FailedToPowerOn; // Error ID to set if command fails
	_strERROR_MSG : T_MaxString		:= 'Failed to power on!'; // Error message to set if command fails
END_VAR
VAR_INST
	_inst_arrParams: T_ApiParameterList; // Parameters array
	_inst_arrOutputs: T_ApiParameterList; // Outputs array
	_inst_strRet: T_ApiParamValue; // Return string from the router
	_inst_intStep: INT; // Current method step
	_inst_fbParams: FB_ApiParamBuilder; // Parameter builder FB
END_VAR
VAR
	_bComplete: BOOL; // True if the routing finishes
	_intRet: INT; // Return string converted to an integer
	_bResult : BOOL; // Output of the method
	_pArgs: PVOID; // Arguments pointer
END_VAR
_bResult := FALSE;

// Recover from premature stop
bPowerOnBusy := TRUE;
_inst_intStep := intPowerOnStep;

// Steps
(* TEMPLATE: Parameters should be added in step 10, and output
	parsing should be added in step 30. *)
CASE _inst_intStep OF
	0: // Wait for no error and router not busy
		IF NOT THIS^.P_bError AND NOT bRouterBusy THEN
			bRouterBusy := TRUE;
			_inst_intStep := _inst_intStep + 10;
		END_IF
		
	10: // Initialize parameters
		THIS^.M_LogMessage(_strSTART_MSG);
		_inst_fbParams.M_ClearParameters();
		_pArgs := _inst_fbParams.M_AddEmptyStruct('args');
		// TEMPLATE: Add any parameters here
		_inst_fbParams.M_OutputToParameterList(_inst_arrParams);
		_inst_intStep := _inst_intStep + 10;
		
	20: // Route the command
		_bComplete := M_RouterHelper(
			_in_strMethodName := _strCOMMAND_NAME, 
			_in_timeTimeout := _timeCOMMAND_TIMEOUT,
			_inout_arrParams := _inst_arrParams,
			_inout_arrOutputs := _inst_arrOutputs,
			_out_strReturnValue=>_inst_strRet);
		
		// If route completed, move to next step
		IF _bComplete THEN
			_inst_intStep := _inst_intStep + 10;
			bRouterBusy := FALSE;
		ELSIF THIS^.P_bError THEN
			_inst_intStep := 0;
			bRouterBusy := FALSE;
		END_IF
		
	30: // Parse results
		_intRet := STRING_TO_INT(_inst_strRet);
		IF _intRet > 0 THEN
			_bResult := TRUE;
			THIS^.M_LogMessage(_strEND_MSG);
			_inst_fbParams.M_LoadFromParameterList(_inst_arrOutputs);
			// TEMPLATE: Do any parsing here
			bPoweredOn := TRUE;
			
		// Set error if command failed
		ELSE
			THIS^.M_SetError(_udintERROR_ID, _strERROR_MSG);
		END_IF
		
		// Go back to start
		_inst_intStep := 0;
END_CASE

M_PowerOn := _bResult;
intPowerOnStep := _inst_intStep;
END_METHOD

(* This property should be TRUE while any method in this interface is actively
	executing, or FALSE otherwise. *)
PROPERTY P_bPowerBusy : BOOL
GET
P_bPowerBusy := bRouterBusy;
END_GET
END_PROPERTY

(* This should be set to TRUE if M_PowerOn is successful or if M_GetPowerStatus
	determines that the device is powered on. Otherwise, this should be FALSE. *)
PROPERTY P_bPoweredOn : BOOL
GET
P_bPoweredOn := bPoweredOn;
END_GET
END_PROPERTY

(* This method should explicitly get the current program loaded on the device.
	If the current program is successfully gotten, this method should return
	TRUE and set P_strCurrentProgram and strCurrentProgram to the gotten
	program name. If this method fails, both should be set to empty strings. *)
METHOD M_GetCurrentProgram : BOOL
VAR_OUTPUT
	(* This should be set to the name of the currently loaded program if
		the method was successful, or a blank string otherwise. *)
	strCurrentProgram	: Sensata_Common.T_MaxString;
END_VAR
VAR CONSTANT
	_strCOMMAND_NAME : T_MaxString	:= 'GetCurrentProgram'; // Name of the API method
	_timeCOMMAND_TIMEOUT : TIME		:= T#10S; // Max time to receive API response
	_strSTART_MSG : T_MaxString		:= 'Getting current program'; // Prints when method starts
	_strEND_MSG : T_MaxString		:= 'Received current program'; // Prints when method finishes
	_udintERROR_ID : UDINT			:= E_ApiDeviceError.FailedToGetCurrentProgram; // Error ID to set if command fails
	_strERROR_MSG : T_MaxString		:= 'Failed to get current program!'; // Error message to set if command fails
END_VAR
VAR_INST
	_inst_arrParams: T_ApiParameterList; // Parameters array
	_inst_arrOutputs: T_ApiParameterList; // Outputs array
	_inst_strRet: T_ApiParamValue; // Return string from the router
	_inst_intStep: INT; // Current method step
	_inst_fbParams: FB_ApiParamBuilder; // Parameter builder FB
END_VAR
VAR
	_bComplete: BOOL; // True if the routing finishes
	_intRet: INT; // Return string converted to an integer
	_bResult : BOOL; // Output of the method
	_pArgs: PVOID; // Arguments pointer
END_VAR
_bResult := FALSE;

// Recover from premature stop
bGetCurrentProgramBusy := TRUE;
_inst_intStep := intGetCurrentProgramStep;

// Steps
(* TEMPLATE: Parameters should be added in step 10, and output
	parsing should be added in step 30. *)
CASE _inst_intStep OF
	0: // Wait for no error and router not busy
		IF NOT THIS^.P_bError AND NOT bRouterBusy THEN
			bRouterBusy := TRUE;
			_inst_intStep := _inst_intStep + 10;
		END_IF
		
	10: // Initialize parameters
		THIS^.M_LogMessage(_strSTART_MSG);
		_inst_fbParams.M_ClearParameters();
		_pArgs := _inst_fbParams.M_AddEmptyStruct('args');
		// TEMPLATE: Add any parameters here
		_inst_fbParams.M_OutputToParameterList(_inst_arrParams);
		_inst_intStep := _inst_intStep + 10;
		
	20: // Route the command
		_bComplete := M_RouterHelper(
			_in_strMethodName := _strCOMMAND_NAME, 
			_in_timeTimeout := _timeCOMMAND_TIMEOUT,
			_inout_arrParams := _inst_arrParams,
			_inout_arrOutputs := _inst_arrOutputs,
			_out_strReturnValue=>_inst_strRet);
		
		// If route completed, move to next step
		IF _bComplete THEN
			_inst_intStep := _inst_intStep + 10;
			bRouterBusy := FALSE;
		ELSIF THIS^.P_bError THEN
			_inst_intStep := 0;
			bRouterBusy := FALSE;
		END_IF
		
	30: // Parse results
		_intRet := STRING_TO_INT(_inst_strRet);
		IF _intRet > 0 THEN
			_bResult := TRUE;
			THIS^.M_LogMessage(_strEND_MSG);
			_inst_fbParams.M_LoadFromParameterList(_inst_arrOutputs);
			// TEMPLATE: Do any parsing here
			THIS^.strLoadedProgram := _inst_fbParams.M_ParseString(
				_inst_fbParams.M_GetParameter('programName'));
			strCurrentProgram := THIS^.strLoadedProgram;
			
		// Set error if command failed
		ELSE
			THIS^.M_SetError(_udintERROR_ID, _strERROR_MSG);
		END_IF
		
		// Go back to start
		_inst_intStep := 0;
END_CASE

M_GetCurrentProgram := _bResult;
intGetCurrentProgramStep := _inst_intStep;
END_METHOD

(* This method should explicitly check the program state of the device.
	Once the program state is known, this method should return TRUE and set
	P_enumProgramState and enumProgramState to the relevant E_ProgramState
	value, else it should set both to E_ProgramState.Unknown. *)
METHOD M_GetProgramState : BOOL
VAR_OUTPUT
	(* If the program state is successfully gotten, this should be set to
		the relevant E_ProgramState value. If this method fails, this should
		be set to E_ProgramState.Unknown. *)
	enumProgramState	: Sensata_Common.E_ProgramState;
END_VAR
VAR CONSTANT
	_strCOMMAND_NAME : T_MaxString	:= 'GetControlState'; // Name of the API method
	_timeCOMMAND_TIMEOUT : TIME		:= T#10S; // Max time to receive API response
	_strSTART_MSG : T_MaxString		:= 'Getting program state'; // Prints when method starts
	_strEND_MSG : T_MaxString		:= 'Received program state'; // Prints when method finishes
	_udintERROR_ID : UDINT			:= E_ApiDeviceError.FailedToGetProgramState; // Error ID to set if command fails
	_strERROR_MSG : T_MaxString		:= 'Failed to get program state!'; // Error message to set if command fails
END_VAR
VAR_INST
	_inst_arrParams: T_ApiParameterList; // Parameters array
	_inst_arrOutputs: T_ApiParameterList; // Outputs array
	_inst_strRet: T_ApiParamValue; // Return string from the router
	_inst_intStep: INT; // Current method step
	_inst_fbParams: FB_ApiParamBuilder; // Parameter builder FB
END_VAR
VAR
	_bComplete: BOOL; // True if the routing finishes
	_intRet: INT; // Return string converted to an integer
	_bResult : BOOL; // Output of the method
	_pArgs: PVOID; // Arguments pointer
	dintControlState: DINT; // Current program state
END_VAR
_bResult := FALSE;

// Recover from premature stop
bGetProgramStateBusy := TRUE;
_inst_intStep := intGetProgramStateStep;

// Steps
(* TEMPLATE: Parameters should be added in step 10, and output
	parsing should be added in step 30. *)
CASE _inst_intStep OF
	0: // Wait for no error and router not busy
		IF NOT THIS^.P_bError AND NOT bRouterBusy THEN
			bRouterBusy := TRUE;
			_inst_intStep := _inst_intStep + 10;
		END_IF
		
	10: // Initialize parameters
		THIS^.M_LogMessage(_strSTART_MSG);
		_inst_fbParams.M_ClearParameters();
		_pArgs := _inst_fbParams.M_AddEmptyStruct('args');
		// TEMPLATE: Add any parameters here
		_inst_fbParams.M_OutputToParameterList(_inst_arrParams);
		_inst_intStep := _inst_intStep + 10;
		
	20: // Route the command
		_bComplete := M_RouterHelper(
			_in_strMethodName := _strCOMMAND_NAME, 
			_in_timeTimeout := _timeCOMMAND_TIMEOUT,
			_inout_arrParams := _inst_arrParams,
			_inout_arrOutputs := _inst_arrOutputs,
			_out_strReturnValue=>_inst_strRet);
		
		// If route completed, move to next step
		IF _bComplete THEN
			_inst_intStep := _inst_intStep + 10;
			bRouterBusy := FALSE;
		ELSIF THIS^.P_bError THEN
			_inst_intStep := 0;
			bRouterBusy := FALSE;
		END_IF
		
